ORGANIZATION_BLOCK "MOD_ERR"	// OB 122
TITLE = "Module Access Error"
AUTHOR : Koenig
VERSION : 0.1
VAR_TEMP
  OB122_EV_CLASS : BYTE ;	//16#29, Event class 2, Entering event state, Internal fault event
  OB122_SW_FLT : BYTE ;	//16#XX Software error code
  OB122_PRIORITY : BYTE ;	//Priority of OB Execution
  OB122_OB_NUMBR : BYTE ;	//122 (Organization block 122, OB122)
  OB122_BLK_TYPE : BYTE ;	//16#88/8C/8E Type of block fault occured in
  OB122_MEM_AREA : BYTE ;	//Memory area where access error occured
  OB122_MEM_ADDR : WORD ;	//Memory address where access error occured
  OB122_BLK_NUM : WORD ;	//Block number in which error occured
  OB122_PRG_ADDR : WORD ;	//Program address where error occured
  OB122_DATE_TIME : DATE_AND_TIME ;	//Date and time OB1 started
END_VAR
BEGIN
NETWORK
TITLE =
END_ORGANIZATION_BLOCK

SYMBOL_TABLE
"IDB_Safe_Main"	DB 1	FB 1
"DB_TRO"	DB 2	DB 2
"DB_LIF"	DB 3	DB 3
"DB_TEL"	DB 4	DB 4
"DB_BRI"	DB 5	DB 5
"DB_ComGateway"	DB 10	DB 10
"IDB_FB2_TRO"	DB 12	FB 2
"IDB_FB2_LIF"	DB 13	FB 2
"IDB_FB21_TEL"	DB 14	FB 21
"DB_OrderBuffer"	DB 15	DB 15
"DB_IntentData"	DB 17	DB 17
"DB_TargetData"	DB 19	DB 19
"IDB_FB22"	DB 22	FB 22
"IDB_FB29"	DB 29	FB 29
"IDB_MasterInterface"	DB 33	FB 13
"DB_ANALOG"	DB 50	DB 50
"INOUT"	DB 80	DB 80
"DB_ActualHookdata"	DB 92	DB 92	// Hookdata of actual trollayposition
"Moves"	DB 101	DB 101
"InstanzDB PNIODiag"	DB 126	FB 126
"InstanzDB STATDiag"	DB 127	DB 127
"DB_Crane"	DB 130	DB 130
"DB_Steps"	DB 132	DB 132
"DB_CylinderTypes"	DB 133	DB 133
"DB_Area"	DB 150	DB 150
"IDB_FB190"	DB 190	FB 190
"IDB_FB190_2"	DB 191	FB 190
"IDB1_FB192"	DB 192	FB 192
"IDB1_FB192_2"	DB 193	FB 192
"TRO_Positions"	DB 200	DB 200
"BR01_TR01"	DB 201	DB 201
"BR01_TR02"	DB 202	DB 202
"BR01_TR03"	DB 203	DB 203
"BR01_TR04"	DB 204	DB 204
"BR01_TR05"	DB 205	DB 205
"BR01_TR06"	DB 206	DB 206
"BR01_TR07"	DB 207	DB 207
"BR01_TR08"	DB 208	DB 208
"BR01_TR09"	DB 209	DB 209
"BR01_TR10"	DB 210	DB 210
"BR01_TR11"	DB 211	DB 211
"BR02_TR01"	DB 212	DB 212
"BR02_TR02"	DB 213	DB 213
"BR02_TR03"	DB 214	DB 214
"BR02_TR04"	DB 215	DB 215
"BR02_TR05"	DB 216	DB 216
"BR02_TR06"	DB 217	DB 217
"BR02_TR07"	DB 218	DB 218
"BR02_TR08"	DB 219	DB 219
"BR02_TR09"	DB 220	DB 220
"BR02_TR10"	DB 221	DB 221
"BR02_TR11"	DB 222	DB 222
"BR03_TR01"	DB 223	DB 223
"BR03_TR02"	DB 224	DB 224
"BR03_TR03"	DB 225	DB 225
"BR03_TR04"	DB 226	DB 226
"BR03_TR05"	DB 227	DB 227
"BR03_TR06"	DB 228	DB 228
"BR03_TR07"	DB 229	DB 229
"BR03_TR08"	DB 230	DB 230
"BR03_TR09"	DB 231	DB 231
"BR03_TR10"	DB 232	DB 232
"BR03_TR11"	DB 233	DB 233
"BR04_TR01"	DB 234	DB 234
"BR04_TR02"	DB 235	DB 235
"BR04_TR03"	DB 236	DB 236
"BR04_TR04"	DB 237	DB 237
"BR04_TR05"	DB 238	DB 238
"BR04_TR06"	DB 239	DB 239
"BR04_TR07"	DB 240	DB 240
"BR04_TR08"	DB 241	DB 241
"BR04_TR09"	DB 242	DB 242
"BR04_TR10"	DB 243	DB 243
"BR04_TR11"	DB 244	DB 244
"BR05_TR01"	DB 245	DB 245
"BR05_TR02"	DB 246	DB 246
"BR05_TR03"	DB 247	DB 247
"BR05_TR04"	DB 248	DB 248
"BR05_TR05"	DB 249	DB 249
"BR05_TR06"	DB 250	DB 250
"BR05_TR07"	DB 251	DB 251
"BR05_TR08"	DB 252	DB 252
"BR05_TR09"	DB 253	DB 253
"BR05_TR10"	DB 254	DB 254
"BR05_TR11"	DB 255	DB 255
"BR06_TR01"	DB 256	DB 256
"BR06_TR02"	DB 257	DB 257
"BR06_TR03"	DB 258	DB 258
"BR06_TR04"	DB 259	DB 259
"BR06_TR05"	DB 260	DB 260
"BR06_TR06"	DB 261	DB 261
"BR06_TR07"	DB 262	DB 262
"BR06_TR08"	DB 263	DB 263
"BR06_TR09"	DB 264	DB 264
"BR06_TR10"	DB 265	DB 265
"BR06_TR11"	DB 266	DB 266
"BR07_TR01"	DB 267	DB 267
"BR07_TR02"	DB 268	DB 268
"BR07_TR03"	DB 269	DB 269
"BR07_TR04"	DB 270	DB 270
"BR07_TR05"	DB 271	DB 271
"BR07_TR06"	DB 272	DB 272
"BR07_TR07"	DB 273	DB 273
"BR07_TR08"	DB 274	DB 274
"BR07_TR09"	DB 275	DB 275
"BR07_TR10"	DB 276	DB 276
"BR07_TR11"	DB 277	DB 277
"BR08_TR01"	DB 278	DB 278
"BR08_TR02"	DB 279	DB 279
"BR08_TR03"	DB 280	DB 280
"BR08_TR04"	DB 281	DB 281
"BR08_TR05"	DB 282	DB 282
"BR08_TR06"	DB 283	DB 283
"BR08_TR07"	DB 284	DB 284
"BR08_TR08"	DB 285	DB 285
"BR08_TR09"	DB 286	DB 286
"BR08_TR10"	DB 287	DB 287
"BR08_TR11"	DB 288	DB 288
"BR09_TR01"	DB 289	DB 289
"BR09_TR02"	DB 290	DB 290
"BR09_TR03"	DB 291	DB 291
"BR09_TR04"	DB 292	DB 292
"BR09_TR05"	DB 293	DB 293
"BR09_TR06"	DB 294	DB 294
"BR09_TR07"	DB 295	DB 295
"BR09_TR08"	DB 296	DB 296
"BR09_TR09"	DB 297	DB 297
"BR09_TR10"	DB 298	DB 298
"BR09_TR11"	DB 299	DB 299
"BR10_TR01"	DB 300	DB 300
"BR10_TR02"	DB 301	DB 301
"BR10_TR03"	DB 302	DB 302
"BR10_TR04"	DB 303	DB 303
"BR10_TR05"	DB 304	DB 304
"BR10_TR06"	DB 305	DB 305
"BR10_TR07"	DB 306	DB 306
"BR10_TR08"	DB 307	DB 307
"BR10_TR09"	DB 308	DB 308
"BR10_TR10"	DB 309	DB 309
"BR10_TR11"	DB 310	DB 310
"BR11_TR01"	DB 311	DB 311
"BR11_TR02"	DB 312	DB 312
"LIF_Pos"	DB 350	DB 350
"IDB_Modbus1"	DB 362	FB 102
"ProfiNet"	DB 400	DB 400
"Error_Safety"	DB 410	DB 410
"IDB_ESTOP_1"	DB 450	FB 215
"IDB_ESTOP_2"	DB 451	FB 185
"F_GLOBDB"	DB 545	DB 545	// F_: F_Global_Data Block
"F00035_4FDI_4FDO_iPar__"	DB 555	FB 272
"F00040_4FDI_4FDO_iPar__"	DB 556	FB 272
"F00045_4FDI_iPar___UINT8"	DB 557	FB 272
"F00055_75x_667_4FDI_4FDO"	DB 558	FB 272
"F_IO"	DB 690	DB 690
"F_Position"	DB 695	DB 695
"F_GBL_RECV"	DB 750	DB 750
"IDB_F_RCV"	DB 751	FB 226
"F_GBL_SEND"	DB 752	DB 752
"IDB_F_SND"	DB 753	FB 225
"IDB_Axis_Position"	DB 800	FB 5
"IDB_WagoiPar_Rack"	DB 901	FB 37
"IDB_WagoiPar_BRI"	DB 920	FB 37
"IDB_WagoiPar_TRO"	DB 921	FB 37
"IDB_WagoiPar_LIF"	DB 922	FB 37
"DB_iPar_Diag"	DB 930	FB 101
"DIAG_PROFI_V2_iPar"	DB 931	DB 931	// diagnosis data of PROFIsafe modules V2 iPar with FB101
"DB_Vorlage"	DB 999	DB 999
"DB_LS1"	DB 1300	DB 1300
"IDB_LS1_Circum"	DB 1329	FB 29
"DB_LS"	DB 1350	DB 1350
"iPar_Data_Rack"	DB 1901	DB 1901
"iPar_Data_Bridge"	DB 1920	DB 1920
"iPar_Data_Trolley"	DB 1921	DB 1921
"iPar_Data_Lift"	DB 1922	DB 1922
"Safe_Main"	FB 1	FB 1
"MovidriveB_Control"	FB 2	FB 2
"Axis_Position"	FB 5	FB 5
"MasterInterface"	FB 13	FB 13
"CheckEncoder"	FB 21	FB 21
"GetCircumference"	FB 22	FB 22
"WAGO_Analog_Input_4_20"	FB 29	FB 29	// WAGO A/D-Wandler 4-20mA
"WAGO_iPar_UDL_4_Mod"	FB 37	FB 37	// WAGO up- / download iParameter PROFIsafe Modules
"TSEND"	FB 63	FB 63	// Send Data
"TRCV"	FB 64	FB 64	// Receive Data
"TCON"	FB 65	FB 65	// Connect
"TDISCON"	FB 66	FB 66	// Disconnect
"Safety_Position"	FB 70	FB 70	// Sichere Positionsüberwachung
"Safety_Direction"	FB 72	FB 72	// Sichere Richtungserfassung
"Safety_Speed"	FB 73	FB 73	// Sichere Geschwindigkeit
"Safety_SpeedCheck"	FB 74	FB 74
"Wago_Trolley"	FB 81	FB 81
"F_Input_MAP"	FB 91	FB 91
"ESTOP"	FB 92	FB 92
"GetArea"	FB 95	FB 95
"DiagPROFIsafe_V2_iPar"	FB 101	FB 101	// read diagnosis data of PROFIsafe modules V2 iPar
"MODBUSPN"	FB 102	FB 102	// MODBUS PN CPU
"TCP_COMM"	FB 103	FB 103	// TCP Kommunikation
"MOD_CLI"	FB 104	FB 104
"MOD_SERV"	FB 105	FB 105
"PNIODiag"	FB 126	FB 126	// Profibus/DP und Profinet/IO-Diagnose
"STATDiag"	FB 127	FB 127	// Zweitbaustein (PNIODiag)
"F_TON"	FB 185	FB 185	// F_: Timer Switch On Delay
"F_TOF"	FB 186	FB 186	// F_: Timer Switch Off Delay
"CopyHookDBs"	FB 190	FB 190
"READ_DBL"	FB 192	FB 192	// read db from memorycard
"WRITE_DBL"	FB 193	FB 193	// write db to memorycard
"F_ESTOP1"	FB 215	FB 215	// F_: Emergency Stop / Stop Category 1
"F_ACK_GL"	FB 219	FB 219	// F_: Global Acknowledgement of all F-I/O of a RTG
"F_SENDS7"	FB 225	FB 225	// F_: Send S7 Connection
"F_RCVS7"	FB 226	FB 226	// F_: Receive S7 Connection
"F_IO_CGP"	FB 272	FB 272	// F_: Driver Block In-Output with Channel Granular Passivation
"F_CTRL_1"	FB 273	FB 273
"F_CTRL_2"	FB 274	FB 274	// F_: Test Block an Programm Run Control
"F_DIAG_N"	FB 275	FB 275
"FITON"	FB 276	FB 276
"FITOF"	FB 277	FB 277
"FIACK_GL"	FB 278	FB 278
"F-CALL"	FC 1	FC 1
"Init"	FC 2	FC 2
"AG_SEND"	FC 5	FC 5	// AG SEND
"AG_RECV"	FC 6	FC 6	// AG RECEIVE
"DT_TOD"	FC 8	FC 8	// DT to TOD
"OpHours"	FC 9	FC 9
"EQ_STRNG"	FC 10	FC 10	// Equal String
"AbsEncoder"	FC 11	FC 11
"Motor_2_frequ"	FC 12	FC 12
"DT to DATE"	FC 15	FC 15	// DT to DATE
"Scan_BRI"	FC 21	FC 21
"Scan_BRI_MAN"	FC 22	FC 22	// Scan Bride Manual Mode
"Scan_BRI_DBs"	FC 23	FC 23
"Scan_LIF"	FC 25	FC 25
"Scan_LIF_Man"	FC 26	FC 26
"Scan_TEL"	FC 27	FC 27
"Scan_TEL_Man"	FC 28	FC 28
"SCALE_WAGO_AI"	FC 29	FC 29	// for WAGO 250-466 4-20mA SE Standard
"Inputs"	FC 30	FC 30
"Outputs"	FC 31	FC 31
"MeasureSystem"	FC 33	FC 33
"SEL"	FC 36	FC 36	// Select
"Errors"	FC 40	FC 40
"Errors Reset"	FC 41	FC 41
"Errors_001-016_GEN1"	FC 42	FC 42
"Errors_017-032_GEN2"	FC 43	FC 43
"Errors_033-048_NET"	FC 44	FC 44
"Errors_113-128"	FC 45	FC 45
"Errors_129-144_08"	FC 46	FC 46
"Errors_145-160"	FC 47	FC 47
"EOff_MachineOff"	FC 48	FC 48
"OP_Mode"	FC 49	FC 49
"Send_Buffer"	FC 52	FC 52
"MSG_161-176"	FC 55	FC 55
"MSG_177_192"	FC 56	FC 56
"CableDrum"	FC 60	FC 60
"TargetPosLift"	FC 70	FC 70
"CheckHookType"	FC 72	FC 72
"CheckWindowDi"	FC 100	FC 100
"Communication"	FC 103	FC 103
"STEPS_Control"	FC 110	FC 110
"STEPS_OrderData"	FC 111	FC 111
"STEPS_BASEPOS"	FC 112	FC 112
"STEPS_EMPTY"	FC 113	FC 113
"STEPS_GET"	FC 114	FC 114
"STEPS_PUT"	FC 115	FC 115
"Axis_TROLLEY"	FC 210	FC 210
"Axis_TROLLEY_Release"	FC 211	FC 211
"Axis_TROLLEY_Control"	FC 212	FC 212
"Axis_TROLLEY_Speed"	FC 213	FC 213
"Axis_TROLLEY_Scan"	FC 214	FC 214
"Axis_TROLLEY_Scan_Man"	FC 215	FC 215
"Axis_TROLLEY_Flt_065-080"	FC 219	FC 219
"Axis_LIFT"	FC 220	FC 220
"Axis_LIFT_Control"	FC 222	FC 222
"Axis_LIFT_Speed"	FC 223	FC 223
"Axis_LIFT_Scan"	FC 224	FC 224
"Axis_LIFT_Flt_081-096"	FC 229	FC 229
"Axis_TELESCOPES"	FC 230	FC 230
"Axis_TEL_Control"	FC 232	FC 232
"Axis_TEL_Speed"	FC 233	FC 233
"Axis_TEL_Scan"	FC 234	FC 234
"Axis_TEL_Chk"	FC 235	FC 235
"Axis_TEL_Status"	FC 236	FC 236
"Axis_TEL_Mode_Status"	FC 237	FC 237
"Axis_TEL_BCD"	FC 238	FC 238
"Axis_TEL_Flt_097-112"	FC 239	FC 239
"Axis_TEL_Encoder"	FC 240	FC 240
"iPar_ServerCall"	FC 900	FC 900
"Scan_LIF_New"	FC 1025	FC 1025
"Scan_LIF_Man_New"	FC 1026	FC 1026
"TROGetPosVal"	FC 1071	FC 1071
"E   35.0"	I 35.0	BOOL	// spare
"E   35.1"	I 35.1	BOOL	// spare
"I_TRO_FB_Lift"	I 35.2	BOOL	// Feedback safestop lift
"I_TRO_FB_Trolley"	I 35.3	BOOL	// Feedback safestop  trolley
"I_TRO_FB_Telescope"	I 40.0	BOOL	// Feedback safestop no FU
"E   40.1"	I 40.1	BOOL	// spare
"I_TRO_FB_Estop_CH1"	I 40.2	BOOL	// Feedback E-Stop  CH1
"I_TRO_FB_Estop_CH2"	I 40.3	BOOL	// Feedback E-Stop  CH2
"I_TRO_EStop"	I 45.0	BOOL	// Emergency stop activ
"I_TRO_Brake_OK"	I 45.1	BOOL	// Temperature brake resistors OK
"E   45.2"	I 45.2	BOOL	// spare
"E   45.3"	I 45.3	BOOL	// spare
"I_TRO_LIF_Overl_L_NC"	I 55.0	BOOL	// Overload-Monitoring left NC
"I_TRO_LIF_Overl_R_NC"	I 55.1	BOOL	// Overload-Monitoring right NC
"I_TRO_LIF_Slap_L_NC"	I 55.2	BOOL	// Slap-Rope-Monitoring left NC
"I_TRO_LIF_Slap_R_NC"	I 55.3	BOOL	// Slap-Rope-Monitoring right NC
"I_TRO_Fuse_115V_OK"	I 75.0	BOOL	// 115V AC OK
"I_TRO_Fuse_24V_OK"	I 75.1	BOOL	// fuse 24V DC OK
"I_TRO_Overtemp_Cabinet"	I 75.2	BOOL	// high temperature cabinet
"I_TRO_Power Brakes_OK"	I 75.3	BOOL	// Power supply brakes OK
"I_TRO_Power_Lift_OK"	I 75.4	BOOL	// Power supply lift OK
"I_TRO_Power_Drum_OK"	I 75.5	BOOL	// Power supply cable drum OK
"I_TRO_Power_Cabinet_Fan"	I 75.6	BOOL	// Power supply cabinet fan OK
"I_TRO_Cabinet_Fan_On"	I 75.7	BOOL	// cabinet fan running
"I_TRO_BTN_Reset"	I 76.0	BOOL	// Reset button (top cabinet)
"I_TRO_BTN_Preset"	I 76.1	BOOL	// Preset button (3s)
"I_TRO_Preset_Bit_0"	I 76.2	BOOL	// Preset selection switch bit 0
"I_TRO_Preset_Bit_1"	I 76.3	BOOL	// Preset selection switch bit 1
"I_TRO_Preset_Bit_2"	I 76.4	BOOL	// Preset selection switch bit 2
"I_TRO_Preset_Bit_3"	I 76.5	BOOL	// Preset selection switch bit 3
"E 76_6"	I 76.6	BOOL	// spare
"E 76_7"	I 76.7	BOOL	// spare
"I_Check_CableDrum_NO"	I 77.0	BOOL	// check cable drum NO
"I_Check_CableDrum_NC"	I 77.1	BOOL	// check cable drum NC
"E  77_2"	I 77.2	BOOL	// spar
"E  77_3"	I 77.3	BOOL	// spar
"I_Buffer_left_Free"	I 77.4	BOOL	// Buffer left occupied //
"I_Buffer_right_Free"	I 77.5	BOOL	// Buffer right occupied //
"I_LIF_Limit_TOP"	I 77.6	BOOL	// Lift limit switch top (minus)
"I_LIF_Limit_BOTTOM"	I 77.7	BOOL	// Lift limit switch bottom (plus)
"I_LIF_Pos_TOP_NO"	I 78.0	BOOL	// Lift limit prox. top NO
"I_LIF_Pos_TOP_NC"	I 78.1	BOOL	// Lift limit prox. top NC
"I_TRO_Limit_plus"	I 78.2	BOOL	// Tolley limit switch plus
"I_TRO_Limit_minus"	I 78.3	BOOL	// Tolley limit switch minus
"I_TRO_FS_plus_NO"	I 78.4	BOOL	// Tolley prox. switch forced slow plus NO
"I_TRO_FS_plus_NC"	I 78.5	BOOL	// Tolley prox. switch forced slow plus NC
"I_TRO_FS_minus_NO"	I 78.6	BOOL	// Tolley prox. switch forced slow minus NO
"I_TRO_FS_minus_NC"	I 78.7	BOOL	// Tolley prox. switch forced slow minus NC
"I_SSI_Barcode_noPos"	I 79.0	BOOL	// Datamatrix SSI error: no position
"I_SSI_Barcode_dirty"	I 79.1	BOOL	// Datamatrix SSI error: dirty
"I_Profinet_Barcode_noPos"	I 79.2	BOOL	// Datamatrix Profinet error: no position
"I_Profinet_Barcode_dirty"	I 79.3	BOOL	// Datamatrix Profinet error: dirty
"I_TRO_Drop_1_P"	I 79.4	BOOL	// Trolley drop off protection plus 1
"I_TRO_Drop_2_P"	I 79.5	BOOL	// Trolley drop off protection plus 2
"I_TRO_Drop_1_M"	I 79.6	BOOL	// Trolley drop off protection minus 1
"I_TRO_Drop_2_M"	I 79.7	BOOL	// Trolley drop off protection minus 2
"I_TRO_Plus"	I 80.0	BOOL	// Trolley drive plus
"I_TRO_Minus"	I 80.1	BOOL	// Trolley drive minus
"I_Lift_up"	I 80.2	BOOL	// Lift drive up
"I_Lift_down"	I 80.3	BOOL	// Lift drive down
"I_TEL_Plus"	I 80.4	BOOL	// Tellescope drive plus
"I_TEL_Minus"	I 80.5	BOOL	// Telescope drive minus
"E 80_6"	I 80.6	BOOL	// spare
"E 80_7"	I 80.7	BOOL	// spare
"E 85_0"	I 85.0	BOOL	// spare
"E 85_1"	I 85.1	BOOL	// spare
"E 85_2"	I 85.2	BOOL	// spare
"E 85_3"	I 85.3	BOOL	// spare
"I_TEL_Status1"	I 85.4	BOOL	// Drive telescopes status1
"I_TEL_Status2"	I 85.5	BOOL	// Drive telescopes status2
"E 85_6"	I 85.6	BOOL
"E 85_7"	I 85.7	BOOL
"I_LIF_Overload_L_NO"	I 86.0	BOOL	// Overload-Monitoring left NO
"I_LIF_Overload_R_NO"	I 86.1	BOOL	// Overload-Monitoring right NO
"I_LIF_SlapRope_L_NO"	I 86.2	BOOL	// Slap-Rope-Monitoring left NO
"I_LIF_SlapRope_R_NO"	I 86.3	BOOL	// Slap-Rope-Monitoring right NO
"E      86.4"	I 86.4	BOOL	// spare
"E      86.5"	I 86.5	BOOL	// spare
"I_LIF_Front_LastHookOcc"	I 86.6	BOOL	// hook front left occupied long
"I_LIF_Front_FirstHookOcc"	I 86.7	BOOL	// hook rear left occupied short
"I_LIF_Rear_LastHookOcc"	I 87.0	BOOL	// hook front right occupied long
"I_LIF_Rear_FirstHookOcc"	I 87.1	BOOL	// hook rear right occupied short
"E      87.2"	I 87.2	BOOL	// spare
"E      87.3"	I 87.3	BOOL	// spare
"I_TEL_inMidle_L"	I 87.4	BOOL	// telescope left in middle position
"I_TEL_inMidle_R"	I 87.5	BOOL	// telescope right in middle position
"E      87.6"	I 87.6	BOOL
"I_TEL_Left_Occ_NO"	I 87.7	BOOL	// telescope left occupied NO
"E      88.0"	I 88.0	BOOL
"I_TEL_Right_Occ_NO"	I 88.1	BOOL	// telescope right occupied NO
"I_TEL_Limit_front_NO"	I 88.2	BOOL	// telescopes limit switch front NO
"I_TEL_Limit_front_NC"	I 88.3	BOOL	// telescopes limit switch front NC
"I_TEL_Limit_back_NO"	I 88.4	BOOL	// telescopes limit switch back NO
"I_TEL_Limit_back_NC"	I 88.5	BOOL	// telescopes limit switch back NC
"E      88.6"	I 88.6	BOOL	// spare
"E      88.7"	I 88.7	BOOL	// spare
"E      89.0"	I 89.0	BOOL
"E      89.1"	I 89.1	BOOL
"E      89.2"	I 89.2	BOOL
"E      89.3"	I 89.3	BOOL
"E      89.4"	I 89.4	BOOL
"E      89.5"	I 89.5	BOOL
"E      89.6"	I 89.6	BOOL
"E      89.7"	I 89.7	BOOL
"OFF"	M 0.0	BOOL	// immer aus
"ON"	M 0.1	BOOL	// immer ein
"FIRST_RUN"	M 0.7	BOOL
"ModeService"	M 1.0	BOOL
"ModeManual"	M 1.1	BOOL
"ModeAuto"	M 1.2	BOOL
"ModeBypass"	M 1.3	BOOL
"ModeServiceOrManual"	M 1.4	BOOL
"SEW_EmergencyMode"	M 1.5	BOOL
"ModeAutoOrManual"	M 1.6	BOOL
"LifeBitMasterOK"	M 1.7	BOOL
"Eoff"	M 2.0	BOOL
"DivEoff"	M 2.1	BOOL
"Error"	M 2.2	BOOL
"EmOffRelais_delayed"	M 3.0	BOOL
"TRO_pFL_StopOnCarrier"	M 8.0	BOOL
"TRO_StopOnCarrier"	M 8.1	BOOL
"LIF_pFl_manPrevPos"	M 9.0	BOOL
"LIF_pFl_manNextPos"	M 9.1	BOOL
"Tel_pFl_manMinusPos"	M 9.2	BOOL
"Tel_pFl_manPlusPos"	M 9.3	BOOL
"TEL_nFl_CenterPos"	M 9.4	BOOL
"TEL_StopInCenter"	M 9.5	BOOL
"TEL_pFl_StopInCenter"	M 9.6	BOOL
"Clock0_1"	M 10.0	BOOL	// CPU-Takt 0,1s
"Clock0_2"	M 10.1	BOOL	// CPU-Takt 0,2s
"Clock0_4"	M 10.2	BOOL	// CPU-Takt 0,4s
"Clock0_5"	M 10.3	BOOL	// CPU-Takt 0,5s
"Clock0_8"	M 10.4	BOOL	// CPU-Takt 0,8s
"Clock1_0"	M 10.5	BOOL	// CPU-Takt 1,0s
"Clock1_6"	M 10.6	BOOL	// CPU-Takt 1,6s
"Clock2_0"	M 10.7	BOOL	// CPU-Takt 2,0s
"Tick0_1"	M 11.0	BOOL	// Impuls 0,1s
"Tick0_2"	M 11.1	BOOL	// Impuls 0,2s
"Tick0_4"	M 11.2	BOOL	// Impuls 0,4s
"Tick0_5"	M 11.3	BOOL	// Impuls 0,6s
"Tick0_8"	M 11.4	BOOL	// Impuls 0,8s
"Tick1_0"	M 11.5	BOOL	// Impuls 1,0s
"Tick1_6"	M 11.6	BOOL	// Impuls 1,6s
"Tick2_0"	M 11.7	BOOL	// Impuls 2,0s
"SysPulse_0_1"	M 12.0	BOOL
"SysPulse_0_2"	M 12.1	BOOL
"SysPulse_0_4"	M 12.2	BOOL
"SysPulse_0_5"	M 12.3	BOOL
"SysPulse_0_8"	M 12.4	BOOL
"SysPulse_1_0"	M 12.5	BOOL
"SysPulse_1_6"	M 12.6	BOOL
"SysPulse_2_0"	M 12.7	BOOL
"StartModeAuto"	M 13.0	BOOL
"TEL_pFl_Start"	M 19.0	BOOL
"NullBit"	M 20.0	BOOL
"CB_Lamp_Preset"	M 21.0	BOOL
"TEL_Save_Long_POS_front"	M 25.0	BOOL
"TEL_Save_Long_POS_rear"	M 25.1	BOOL
"TrolleyWasOnCarrier"	M 40.0	BOOL
"SendTrolleyWasOnCarrier"	M 40.1	BOOL
"Next_Step"	M 44.0	BOOL
"SingleStep_ON"	M 44.1	BOOL
"One_Single_Step"	M 44.2	BOOL
"TEL_RackPos"	M 55.0	BOOL
"TEL_LS1_Pos"	M 55.1	BOOL
"TEL_LS2_Pos"	M 55.2	BOOL
"TEL_LS3_Pos"	M 55.3	BOOL
"Safety_Tele_Center"	M 152.0	BOOL
"Safety_Tele_Rear"	M 152.1	BOOL
"Safety_Tele_Front"	M 152.2	BOOL
"Safety_Trolley_in_Pos"	M 153.0	BOOL
"Safety_Lift_Top"	M 154.0	BOOL
"Safety_Lift_Over"	M 154.1	BOOL
"Safety_Lift_Under"	M 154.2	BOOL
"Mode_Bypass"	M 200.2	BOOL
"RED_IBN_Test"	M 420.0	BOOL
"TRUE"	M 500.0	BOOL
"FALSE"	M 500.1	BOOL
"IBN_1"	M 501.0	BOOL
"IBN_0"	M 501.1	BOOL
"IBN_Test"	M 501.2	BOOL
"TRO_iPar_Check"	M 921.0	BOOL
"TRO_iPar_UpLoad"	M 921.1	BOOL
"TRO_iPar_DownL"	M 921.2	BOOL
"TRO_iPar_ReqDiag"	M 921.5	BOOL
"LIF_iPar_Check"	M 922.0	BOOL
"LIF_iPar_UpLoad"	M 922.1	BOOL
"LIF_iPar_DownL"	M 922.2	BOOL
"LIF_iPar_ReqDiag"	M 922.5	BOOL
"TRO_pFl_iPar"	M 925.1	BOOL
"LIF_pFl_iPar_1"	M 925.2	BOOL
"LIF_pFl_iPar_2"	M 925.3	BOOL
"PowerFan_pl"	M 1001.0	BOOL
"PowerFan_n"	M 1001.1	BOOL
"P_FL_TeleCheck1"	M 1401.2	BOOL
"N_FL_TeleCheck1"	M 1401.3	BOOL
"P_FL_TeleCheck2"	M 1401.6	BOOL
"N_FL_TeleCheck2"	M 1401.7	BOOL
"TeleCheckErr1"	M 1402.0	BOOL
"TeleCheckErr2"	M 1402.1	BOOL
"TeleCheckErr3"	M 1402.3	BOOL
"TeleCheckErr4"	M 1402.4	BOOL
"Reset_Err"	M 1410.0	BOOL
"Impuls_1"	M 1500.0	BOOL
"Impuls_2"	M 1500.1	BOOL
"Impuls_3"	M 1500.2	BOOL
"Impuls_4"	M 1500.3	BOOL
"Impuls_5"	M 1500.4	BOOL
"Impuls_6"	M 1500.5	BOOL
"Impuls_7"	M 1500.6	BOOL
"Impuls_8"	M 1500.7	BOOL
"TEL_SaveTarget"	MW 14	INT
"NullWord"	MW 20	WORD
"PC_MSG_Counter"	MW 120	INT
"CYCL_EXC"	OB 1	OB 1
"CYC_INT5"	OB 35	OB 35	// Cyclic Interrupt 5
"CYCL_FLT"	OB 80	OB 80	// Cycle Time Fault
"I/O_FLT1"	OB 82	OB 82	// I/O Point Fault 1
"I/O_FLT2"	OB 83	OB 83	// I/O Point Fault 2
"OBNL_FLT"	OB 85	OB 85	// OB Not Loaded Fault
"RACK_FLT"	OB 86	OB 86	// Loss of Rack Fault
"COMM_FLT"	OB 87	OB 87	// Communication Fault
"STARTUP"	OB 100	OB 100
"PROG_ERR"	OB 121	OB 121	// Programming Error
"MOD_ERR"	OB 122	OB 122	// Module Access Error
"O_Bypass_RC"	Q 35.0	BOOL	// bypass remote control
"A    35.1"	Q 35.1	BOOL	// spare
"O_SafeStop_Lift"	Q 35.2	BOOL	// safe stop lift
"O_SafeStop_Trolley"	Q 35.3	BOOL	// safe stop trolley
"O_SafeStop_Telecope"	Q 40.0	BOOL	// safe stop telescope
"A    40.1"	Q 40.1	BOOL	// spare
"O_TRO_Stop_CH1"	Q 40.2	BOOL	// E-Stop trolley CH1
"O_TRO_Stop_CH2"	Q 40.3	BOOL	// E-Stop trolley CH2
"O_SafeRelease_Telescope"	Q 55.0	BOOL
"A 75_0"	Q 75.0	BOOL	// spare
"O_TRO_Reset_24V"	Q 75.1	BOOL	// reset 24V fuses
"A 75_2"	Q 75.2	BOOL	// spare
"O_TRO_LP_Reset"	Q 75.3	BOOL	// lamp reset
"A 75_4"	Q 75.4	BOOL	// spare
"O_TRO_CableDrum"	Q 75.5	BOOL	// start cable drum
"O_TRO_EStop_Reset"	Q 75.6	BOOL	// ESTOP reset
"O_TRO_LP_Preset"	Q 75.7	BOOL	// lamp preset
"O_TRO_Horn"	Q 76.0	BOOL	// startup warning
"O_TRO_State_0"	Q 76.1	BOOL	// lamp state 0
"O_TRO_State_1"	Q 76.2	BOOL	// lamp state 1
"O_TRO_state_2"	Q 76.3	BOOL	// lamp state 2
"A      76.4"	Q 76.4	BOOL	// spare
"O_TRO_MoviPLC_Reset"	Q 76.5	BOOL	// reset movi PLC
"O_TRO_EmergencyMode"	Q 76.6	BOOL	// Emergency Mode
"O_LIFT_StartFan"	Q 76.7	BOOL	// start Lift Fan
"O_TRO_EmergencyMode_Fwd"	Q 77.0	BOOL	// Emergency mode forward
"O_TRO_EmergencyMode_Bwd"	Q 77.1	BOOL	// Emergency mode backward
"A      77.2"	Q 77.2	BOOL
"A      77.3"	Q 77.3	BOOL
"A      77.4"	Q 77.4	BOOL
"A      77.5"	Q 77.5	BOOL
"A      77.6"	Q 77.6	BOOL
"A      77.7"	Q 77.7	BOOL
"O_TEL_Mode1"	Q 85.0	BOOL	// telescope mode_1 Service
"O_TEL_Mode2"	Q 85.1	BOOL	// telescope mode_2 Automatic
"O_TEL_Start"	Q 85.2	BOOL	// start telescope
"O_TEL_Reset"	Q 85.3	BOOL	// reset telescope
"O_TEL_BCD_Bit_1"	Q 85.4	BOOL	// telescope BCD Bit_1
"O_TEL_BCD_Bit_2"	Q 85.5	BOOL	// telescope BCD Bit_2
"O_TEL_BCD_Bit_3"	Q 85.6	BOOL	// telescope BCD Bit_3
"O_TEL_BCD_Bit_4"	Q 85.7	BOOL	// telescope BCD Bit_4
"O_TEL_LightFront_Left"	Q 86.0	BOOL	// lightning telescopes front left ON
"O_TEL_LightFront_Right"	Q 86.1	BOOL	// lightning telescopes rear rigth ON
"O_TEL_LightRear_Left"	Q 86.2	BOOL	// lightning telescopes rear left ON
"O_TEL_LightRear_Right"	Q 86.3	BOOL	// lightning telescopes rear rigth ON
"O_TEL_Preset_Encoder"	Q 86.4	BOOL	// Preset Encoder Telescope
"A     86.5"	Q 86.5	BOOL	// spare
"A     86.6"	Q 86.6	BOOL	// spare
"A     86.7"	Q 86.7	BOOL	// spare
"A     87.0"	Q 87.0	BOOL
"A     87.1"	Q 87.1	BOOL
"A     87.2"	Q 87.2	BOOL
"A     87.3"	Q 87.3	BOOL
"A     87.4"	Q 87.4	BOOL
"A     87.5"	Q 87.5	BOOL
"A     87.6"	Q 87.6	BOOL
"A     87.7"	Q 87.7	BOOL
"TON"	SFB 4	SFB 4	// Generate an On Delay
"USEND"	SFB 8	SFB 8	// Uncoordinated Sending of Data
"URCV"	SFB 9	SFB 9	// Uncoordinated Receiving of Data
"RDREC"	SFB 52	SFB 52	// Read a Process Data Record
"WRREC"	SFB 53	SFB 53	// Write a Process Data Record
"RALRM"	SFB 54	SFB 54	// Receive Alarm Data
"DPRD_DAT"	SFC 14	SFC 14	// Read Consistent Data of a Standard DP Slave
"DPWR_DAT"	SFC 15	SFC 15	// Write Consistent Data to a Standard DP Slave
"BLKMOV"	SFC 20	SFC 20	// Copy Variables
"FILL"	SFC 21	SFC 21	// Initialize a Memory Area
"TEST_DB"	SFC 24	SFC 24	// Test Data Block
"DIS_AIRT"	SFC 41	SFC 41	// Delay the Higher Priority Interrupts and Asynchronous Errors
"EN_AIRT"	SFC 42	SFC 42	// Enable Higher Priority Interrupts and Asynchronous Errors
"STP"	SFC 46	SFC 46	// Change the CPU to STOP
"RDSYSST"	SFC 51	SFC 51	// Read a System Status List or Partial List
"WR_REC"	SFC 58	SFC 58	// Write Data Record
"RD_REC"	SFC 59	SFC 59	// Read a Data Record
"RD_DBL"	SFC 83	SFC 83	// Read Data Block from Load Memory
"WRIT_DBL"	SFC 84	SFC 84	// Write Data Block in Load Memory
"tPlcOn"	T 1	TIMER
"tAknowl"	T 2	TIMER
"tTimeout_TRO"	T 26	TIMER
"T_TRO_Preset"	T 30	TIMER
"tTimeout_LIF"	T 36	TIMER
"tTimeout_LIF2"	T 37	TIMER
"T_Startup_Warning"	T 94	TIMER
"T_Delay_Emeg_Mode"	T 110	TIMER
"T_Err_TR_Forced_minus"	T 152	TIMER
"T_Err_TR_Forced_plus"	T 153	TIMER
"T_CheckUS"	T 160	TIMER
"T_CheckUS_OK"	T 161	TIMER
"UDT_Any"	UDT 1	UDT 1
"UDT_SysSave"	UDT 2	UDT 2
"OneMove"	UDT 7	UDT 7
"UDT_SEWState"	UDT 11	UDT 11
"UDT_SEWControl"	UDT 12	UDT 12
"TrDataSheet"	UDT 20	UDT 20	// Zuordnung Turm-DBs
"TRODataSheet"	UDT 21	UDT 21
"HookData"	UDT 100	UDT 100
"HookDataSheetNeu"	UDT 101	UDT 101
"HookDataSheet"	UDT 102	UDT 102
"UDT_CylinderType"	UDT 110	UDT 110
"ROW5"	VAT 1	
"IO-Check"	VAT 2	
"ROW4"	VAT 3	
"ROW3"	VAT 4	
"ROW2"	VAT 5	
"ROW1"	VAT 6	
"ROW6"	VAT 7	
"Order"	VAT 8	
"VAT_Sonar"	VAT 9	
"VAT_Bruno"	VAT 10	
"VAT_NewTarget"	VAT 11	
"VAT_TEL_Encoder"	VAT 12	
"VAT_TR_POS_TEST"	VAT 13	
END_SYMBOL_TABLE

TYPE "UDT_Any"	// UDT 1
VERSION : 0.1
  STRUCT
   CONST : BYTE  := B#16#10;	//SIMATIC Constant
   DATATYPE : BYTE ;	//S7-Datatype
   LENGTH : INT ;	//Length of pointer
   DBNO : INT ;	//Datablock Number
   ADDRESS : DWORD ;	//Start address of pointer
  END_STRUCT ;	
END_TYPE

TYPE "UDT_SysSave"	// UDT 2
VERSION : 0.1
  STRUCT
   AR1 : DWORD ;	//adress register 1
   AR2 : DWORD ;	//adress register 2
   DBNO : WORD ;	//DB register
   DINO : WORD ;	//DI register
  END_STRUCT ;	
END_TYPE

TYPE "OneMove"	// UDT 7
VERSION : 0.1
  STRUCT
   MsgCounter : INT ;
   Action : INT ;
   Value_01 : INT ;
   Value_02 : INT ;
   Value_03 : INT ;
   Value_04 : INT ;
   Value_05 : INT ;
   Value_06 : INT ;
   Value_07 : INT ;
   Value_08 : INT ;
   Value_09 : INT ;
   Value_10 : INT ;
   CRC : INT ;
  END_STRUCT ;	
END_TYPE

TYPE "UDT_SEWState"	// UDT 11
VERSION : 0.1
  STRUCT
   State : STRUCT
    Code00 : BOOL ;
    Code01 : BOOL ;
    Code02 : BOOL ;
    Code03 : BOOL ;
    Code04 : BOOL ;
    Code05 : BOOL ;
    Code06 : BOOL ;
    Code07 : BOOL ;
    NgrZero : BOOL ;
    Ready : BOOL ;
    RefOk : BOOL ;
    InPos : BOOL ;
    BrakeOpen : BOOL ;
    ErrWarn : BOOL ;
    LimitRight : BOOL ;
    LimitLeft : BOOL ;
   END_STRUCT ;
   actPosition : DINT ;
   actSpeed : INT ;
   actCurrent : INT ;
   actWorkLoad : INT ;
  END_STRUCT ;	
END_TYPE

TYPE "UDT_SEWControl"	// UDT 12
VERSION : 0.1
  STRUCT
   Control : STRUCT
    Start : BOOL ;
    InchPlus : BOOL ;
    InchMinus : BOOL ;
    Mode11 : BOOL ;
    Mode12 : BOOL ;
    Crt05 : BOOL ;
    Crt06 : BOOL ;
    BypassLimits : BOOL ;
    Lock : BOOL ;
    ReleaseFastStop : BOOL ;
    ReleaseHalt : BOOL ;
    NotPosCrt : BOOL ;
    RampSet2 : BOOL ;
    ParaSet2 : BOOL ;
    Reset : BOOL ;
    Crt17 : BOOL ;
   END_STRUCT ;
   TarPos : DINT ;
   TarSpeed : INT ;
   TarAcc : INT ;
   TarDeac : INT ;
  END_STRUCT ;	
END_TYPE

TYPE "TrDataSheet"	// UDT 20
VERSION : 0.1
  STRUCT
   TroPosVal : DINT ;	//value of trolleyposition
   HookDbNo : INT ;	//number of DB hookdatasheets
  END_STRUCT ;	
END_TYPE

TYPE "TRODataSheet"	// UDT 21
VERSION : 0.1
  STRUCT
   No : INT ;	//number of trolleyposition
   Val : DINT ;	//value of trolleyposition
   HookDbNo : INT ;	//number of DB hookdatasheets
  END_STRUCT ;	
END_TYPE

TYPE "HookData"	// UDT 100
VERSION : 0.1
  STRUCT
   HookType : INT ;
   TotLengthMin : INT ;
   TotLengthMax : INT ;
   FaceLengthMax : INT ;
   CircumMax : INT ;
   TelPos : DINT ;
   Reserve1 : INT ;
  END_STRUCT ;	
END_TYPE

TYPE "HookDataSheetNeu"	// UDT 101
VERSION : 0.1
  STRUCT
   HookOver : DINT ;
   HookUnderOffset : DINT ;
   Telpos_in : DINT ;
   Telpos_mid : DINT ;
   Telpos_out : DINT ;
   TotLengthMin : INT ;
   TotLengthMax : INT ;
   FaceLengthMax : INT ;
   CircumMax : INT ;
   Hooktype : INT ;
   reserve30 : INT ;
  END_STRUCT ;	
END_TYPE

TYPE "HookDataSheet"	// UDT 102
VERSION : 0.1
  STRUCT
   HookOver : DINT ;
   HookUnderOffset : DINT ;
   TelPos_1 : UDT 100;
   TelPos_2 : UDT 100;
   TelPos_3 : UDT 100;
  END_STRUCT ;	
END_TYPE

TYPE "UDT_CylinderType"	// UDT 110
VERSION : 0.1
  STRUCT
   Number : INT ;
   DiameterName : INT ;
   DiameterMin : INT ;
   DiameterMax : INT ;
   Reserve1 : INT ;
  END_STRUCT ;	
END_TYPE

FUNCTION_BLOCK "Safe_Main"	// FB 1
TITLE = Main safety
AUTHOR : Koenig
VERSION : 0.1
VAR
  ON : BOOL ;
  OFF : BOOL ;
  M_Reset : BOOL ;
  M_Automatic : BOOL ;
  StateOK : BOOL ;
  HardwareOK : BOOL ;
  ESTOP : BOOL ;
  ESTOP_DEL : BOOL ;
  Rel_LS : BOOL ;
  Stop_Doors : BOOL ;
  Stop_Doors_DEL : BOOL ;
  Rel_RBG : BOOL ;
  Rel_Trolley : BOOL ;
  Rel_Lift : BOOL ;
  Rel_Telescope : BOOL ;
  ResetGBL : BOOL ;
  RequestGBL : BOOL ;
  SubsGBL : BOOL ;
  Ack : FB 219;
  IO : FB 91;
  E_Stop : FB 92;
  DEL_Doors : FB 185;
  Wago_Trolley_Lift : FB 81;
  TRO_Valid : BOOL ;
  TRO_SafePos : FB 70;
  TRO_SafeAxis : INT ;
  Get_Area : FB 95;
  Difference_Lo : INT ;
  Difference_Hi : INT ;
  TRO_Speed : FB 74;
  TRO_SafeAxis_Speed : INT ;
  TRO_Direction_Plus : BOOL ;
  TRO_Direction_Minus : BOOL ;
  TRO_Direction : FB 72;
  TRO_Direction_Stop : BOOL ;
  Err_SafeSpeed : BOOL ;
  Err_SafeSpeed_Max : BOOL ;
  T_Reset_GBL : FB 185;
  GetArea : FB 95;
END_VAR
BEGIN
// body was compiled from another editor; compiled code not shown
END_FUNCTION_BLOCK

FUNCTION_BLOCK "MovidriveB_Control"	// FB 2
TITLE = MovidriveB_Control
//main control for the SEW controller
//KNOW_HOW_PROTECT 
//
AUTHOR : Koenig
VERSION : 0.1
VAR_INPUT
  StateWord : INT ;
  FastStop : BOOL ;
  Reset : BOOL ;
  Start : BOOL ;
  InchMinus : BOOL ;
  InchPlus : BOOL ;
  ModeService : BOOL ;
  ModeAuto : BOOL ;
  ModeRef : BOOL ;
  Bypass : BOOL ;
  PlcOn : BOOL ;
  Pulse_1_0 : BOOL ;
  Tick_0_1 : BOOL ;
  ActualPosition : DINT ;
  TargetPosition : DINT ;
  TargetPositionNo : INT ;
  LimitPlus : DINT ;
  LimitMinus : DINT ;
  InPosWin : DINT ;
END_VAR
VAR_OUTPUT
  CrtWord : INT ;
  Moves : BOOL ;
  Ready : BOOL ;
  RefOk : BOOL ;
  InPos : BOOL ;
  BrakeOpen : BOOL ;
  Error : BOOL ;
  ErrCode : INT ;
  ActPosition : DINT ;
  ActPositionNo : INT ;
  ActTarget : DINT ;
END_VAR
VAR
  INT_iCntRelHalt : INT ;
  INT_iCntInPos : INT ;
  INT_ActualPosition : DINT ;
  INT_ActualPositionNo : INT ;
  INT_pFl_ResetPosition : BOOL ;
  INT_TargetOK : BOOL ;
END_VAR
VAR_TEMP
  INT_xStateCode00 : BOOL ;
  INT_xStateCode01 : BOOL ;
  INT_xStateCode02 : BOOL ;
  INT_xStateCode03 : BOOL ;
  INT_xStateCode04 : BOOL ;
  INT_xStateCode05 : BOOL ;
  INT_xStateCode06 : BOOL ;
  INT_xStateCode07 : BOOL ;
  INT_xState : BOOL ;
  INT_xStateReady : BOOL ;
  INT_xStateRefOk : BOOL ;
  INT_xStateInPos : BOOL ;
  INT_xStateNgrNull : BOOL ;
  INT_xStateErrWarn : BOOL ;
  INT_xStateLimitRight : BOOL ;
  INT_xStateLimitLeft : BOOL ;
  INT_xCrtStart : BOOL ;
  INT_xCrtInchPlus : BOOL ;
  INT_xCrtInchMinus : BOOL ;
  INT_xCrtMode11 : BOOL ;
  INT_xCrtMode12 : BOOL ;
  INT_xCrt13 : BOOL ;
  INT_xCrt14 : BOOL ;
  INT_xCrtBypassLimits : BOOL ;
  INT_xCrtLock : BOOL ;
  INT_xCrtRelFaststop : BOOL ;
  INT_xCrtRelHalt : BOOL ;
  INT_xCrtNotPosCrt : BOOL ;
  INT_xCrtRampsSet2 : BOOL ;
  INT_xCrtParaSet2 : BOOL ;
  INT_xCrtReset : BOOL ;
  INT_xCrt06 : BOOL ;
  INT_xModeMan : BOOL ;
  INT_xModeAuto : BOOL ;
  INT_xModeRef : BOOL ;
  INT_ON : BOOL ;
  INT_w00 : WORD ;
  mValue : DINT ;
  pValue : DINT ;
END_VAR
BEGIN
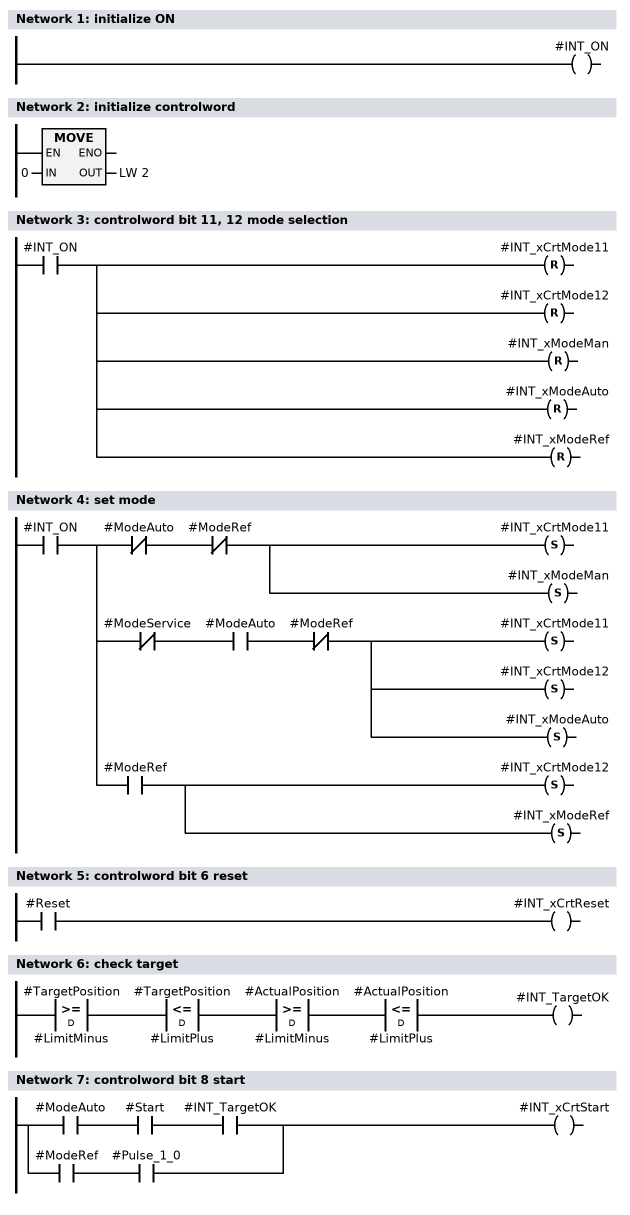
NETWORK
TITLE = initialize ON
//LW0: controler state word
//LW2: controler control word
      SET;
      =     #INT_ON;
NETWORK
TITLE = initialize controlword
      L     0;
      T     LW 2;
      NOP   0;
NETWORK
TITLE = controlword bit 11, 12 mode selection
      A     #INT_ON;
      R     #INT_xCrtMode11;
      R     #INT_xCrtMode12;
      R     #INT_xModeMan;
      R     #INT_xModeAuto;
      R     #INT_xModeRef;
NETWORK
TITLE = set mode
      A     #INT_ON;
      =     L 16.0;
      A     L 16.0;
      AN    #ModeAuto;
      AN    #ModeRef;
      S     #INT_xCrtMode11;
      S     #INT_xModeMan;
      A     L 16.0;
      AN    #ModeService;
      A     #ModeAuto;
      AN    #ModeRef;
      S     #INT_xCrtMode11;
      S     #INT_xCrtMode12;
      S     #INT_xModeAuto;
      A     L 16.0;
      A     #ModeRef;
      S     #INT_xCrtMode12;
      S     #INT_xModeRef;
NETWORK
TITLE = controlword bit 6 reset
      A     #Reset;
      =     #INT_xCrtReset;
NETWORK
TITLE = check target
      A(;
      L     #TargetPosition;
      L     #LimitMinus;
      >=D;
      );
      A(;
      L     #TargetPosition;
      L     #LimitPlus;
      <=D;
      );
      A(;
      L     #ActualPosition;
      L     #LimitMinus;
      >=D;
      );
      A(;
      L     #ActualPosition;
      L     #LimitPlus;
      <=D;
      );
      =     #INT_TargetOK;
NETWORK
TITLE = controlword bit 8 start
      A     #ModeAuto;
      A     #Start;
      A     #INT_TargetOK;
      O;
      A     #ModeRef;
      A     #Pulse_1_0;
      =     #INT_xCrtStart;
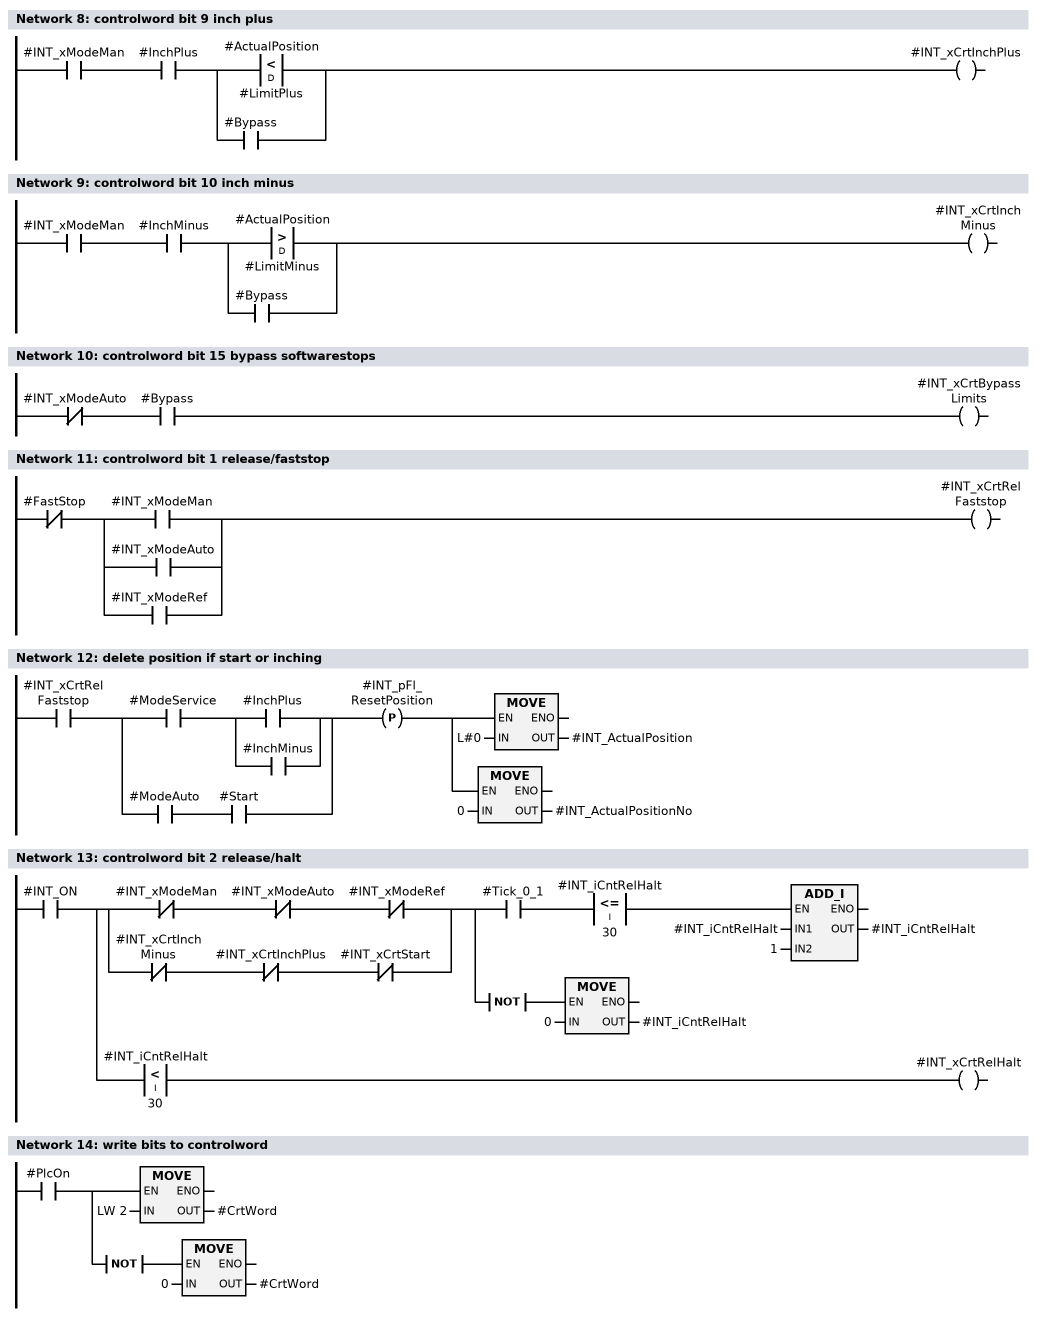
NETWORK
TITLE = controlword bit 9 inch plus
      A     #INT_xModeMan;
      A     #InchPlus;
      A(;
      O(;
      L     #ActualPosition;
      L     #LimitPlus;
      <D;
      );
      O     #Bypass;
      );
      =     #INT_xCrtInchPlus;
NETWORK
TITLE = controlword bit 10 inch minus
      A     #INT_xModeMan;
      A     #InchMinus;
      A(;
      O(;
      L     #ActualPosition;
      L     #LimitMinus;
      >D;
      );
      O     #Bypass;
      );
      =     #INT_xCrtInchMinus;
NETWORK
TITLE = controlword bit 15 bypass softwarestops
      AN    #INT_xModeAuto;
      A     #Bypass;
      =     #INT_xCrtBypassLimits;
NETWORK
TITLE = controlword bit 1 release/faststop
      AN    #FastStop;
      A(;
      O     #INT_xModeMan;
      O     #INT_xModeAuto;
      O     #INT_xModeRef;
      );
      =     #INT_xCrtRelFaststop;
NETWORK
TITLE = delete position if start or inching
      A     #INT_xCrtRelFaststop;
      A(;
      A     #ModeService;
      A(;
      O     #InchPlus;
      O     #InchMinus;
      );
      O;
      A     #ModeAuto;
      A     #Start;
      );
      FP    #INT_pFl_ResetPosition;
      =     L 16.0;
      A     L 16.0;
      JNB   _001;
      L     L#0;
      T     #INT_ActualPosition;
_001: NOP   0;
      A     L 16.0;
      JNB   _002;
      L     0;
      T     #INT_ActualPositionNo;
_002: NOP   0;
NETWORK
TITLE = controlword bit 2 release/halt
      A     #INT_ON;
      =     L 16.0;
      A     L 16.0;
      A(;
      AN    #INT_xModeMan;
      AN    #INT_xModeAuto;
      AN    #INT_xModeRef;
      O;
      AN    #INT_xCrtInchMinus;
      AN    #INT_xCrtInchPlus;
      AN    #INT_xCrtStart;
      );
      =     L 16.1;
      A     L 16.1;
      A     #Tick_0_1;
      A(;
      L     #INT_iCntRelHalt;
      L     30;
      <=I;
      );
      JNB   _003;
      L     #INT_iCntRelHalt;
      L     1;
      +I;
      T     #INT_iCntRelHalt;
_003: NOP   0;
      A     L 16.1;
      NOT;
      JNB   _004;
      L     0;
      T     #INT_iCntRelHalt;
_004: NOP   0;
      A     L 16.0;
      A(;
      L     #INT_iCntRelHalt;
      L     30;
      <I;
      );
      =     #INT_xCrtRelHalt;
NETWORK
TITLE = write bits to controlword
      A     #PlcOn;
      =     L 16.0;
      A     L 16.0;
      JNB   _005;
      L     LW 2;
      T     #CrtWord;
_005: NOP   0;
      A     L 16.0;
      NOT;
      JNB   _006;
      L     0;
      T     #CrtWord;
_006: NOP   0;
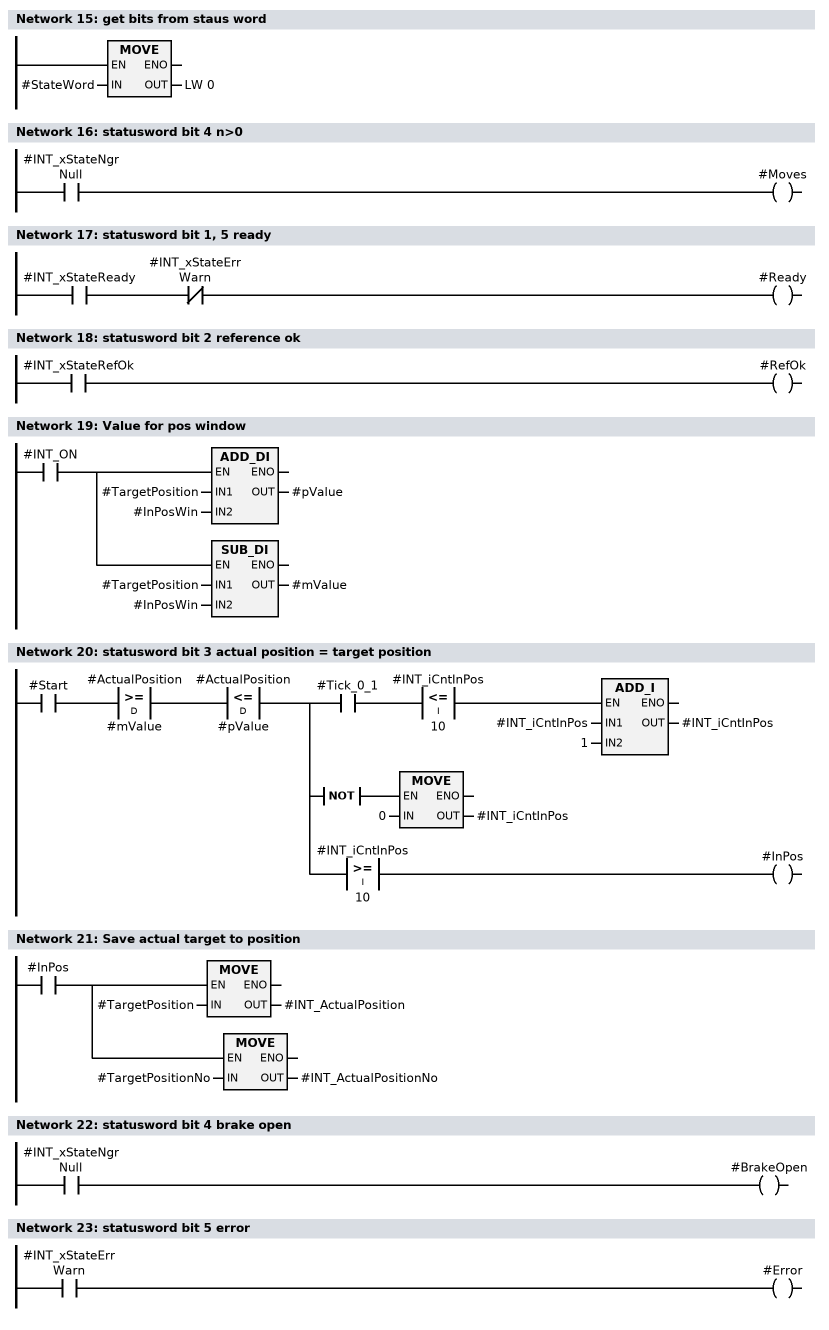
NETWORK
TITLE = get bits from staus word
      L     #StateWord;
      T     LW 0;
      NOP   0;
NETWORK
TITLE = statusword bit 4 n>0
      A     #INT_xStateNgrNull;
      =     #Moves;
NETWORK
TITLE = statusword bit 1, 5 ready
      A     #INT_xStateReady;
      AN    #INT_xStateErrWarn;
      =     #Ready;
NETWORK
TITLE = statusword bit 2 reference ok
      A     #INT_xStateRefOk;
      =     #RefOk;
NETWORK
TITLE = Value for pos window
      A     #INT_ON;
      =     L 16.0;
      A     L 16.0;
      JNB   _007;
      L     #TargetPosition;
      L     #InPosWin;
      +D;
      T     #pValue;
_007: NOP   0;
      A     L 16.0;
      JNB   _008;
      L     #TargetPosition;
      L     #InPosWin;
      -D;
      T     #mValue;
_008: NOP   0;
NETWORK
TITLE = statusword bit 3 actual position = target position
//note: in omron we use the actual position and the target postion equal
//
      A     #Start;
      A(;
      L     #ActualPosition;
      L     #mValue;
      >=D;
      );
      A(;
      L     #ActualPosition;
      L     #pValue;
      <=D;
      );
      =     L 16.0;
      A     L 16.0;
      A     #Tick_0_1;
      A(;
      L     #INT_iCntInPos;
      L     10;
      <=I;
      );
      JNB   _009;
      L     #INT_iCntInPos;
      L     1;
      +I;
      T     #INT_iCntInPos;
_009: NOP   0;
      A     L 16.0;
      NOT;
      JNB   _00a;
      L     0;
      T     #INT_iCntInPos;
_00a: NOP   0;
      A     L 16.0;
      A(;
      L     #INT_iCntInPos;
      L     10;
      >=I;
      );
      =     #InPos;
NETWORK
TITLE = Save actual target to position
      A     #InPos;
      =     L 16.0;
      A     L 16.0;
      JNB   _00b;
      L     #TargetPosition;
      T     #INT_ActualPosition;
_00b: NOP   0;
      A     L 16.0;
      JNB   _00c;
      L     #TargetPositionNo;
      T     #INT_ActualPositionNo;
_00c: NOP   0;
NETWORK
TITLE = statusword bit 4 brake open
      A     #INT_xStateNgrNull;
      =     #BrakeOpen;
NETWORK
TITLE = statusword bit 5 error
      A     #INT_xStateErrWarn;
      =     #Error;
NETWORK
TITLE = status / error code
      A     #INT_ON;
      =     L 16.0;
      A     L 16.0;
      JNB   _00d;
      L     LW 0;
      L     W#16#FF00;
      AW;
      T     LW 0;
_00d: NOP   0;
      A     L 16.0;
      JNB   _00e;
      L     W#16#8;
      L     LW 0;
      SRW;
      T     LW 0;
_00e: NOP   0;
      A     L 16.0;
      JNB   _00f;
      L     LW 0;
      T     #ErrCode;
_00f: NOP   0;
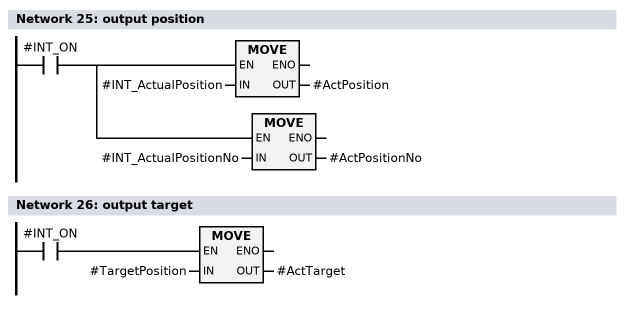
NETWORK
TITLE = output position
      A     #INT_ON;
      =     L 16.0;
      A     L 16.0;
      JNB   _010;
      L     #INT_ActualPosition;
      T     #ActPosition;
_010: NOP   0;
      A     L 16.0;
      JNB   _011;
      L     #INT_ActualPositionNo;
      T     #ActPositionNo;
_011: NOP   0;
NETWORK
TITLE = output target
      A     #INT_ON;
      JNB   _012;
      L     #TargetPosition;
      T     #ActTarget;
_012: NOP   0;
END_FUNCTION_BLOCK

FUNCTION_BLOCK "Axis_Position"	// FB 5
TITLE = Axis_Position
AUTHOR : BRO
VERSION : 0.1
VAR_INPUT
  Inpos : DINT ;
END_VAR
VAR_OUTPUT
  OutPos : DINT ;
END_VAR
BEGIN
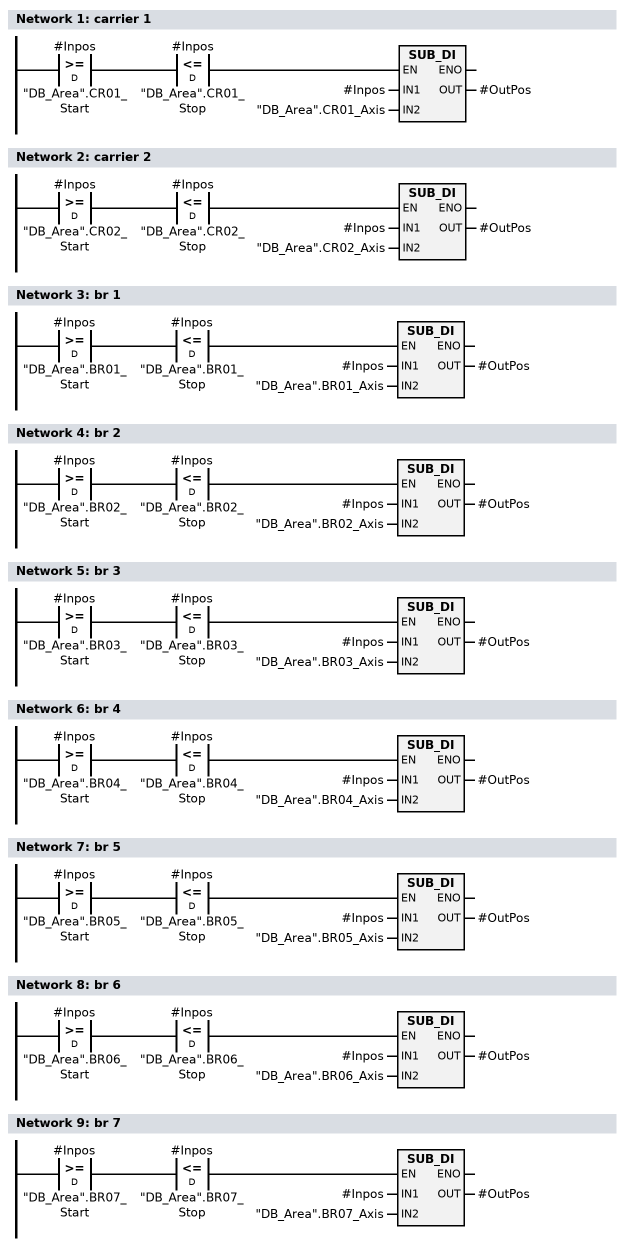
NETWORK
TITLE = carrier 1
      A(;
      L     #Inpos;
      L     "DB_Area".CR01_Start;
      >=D;
      );
      A(;
      L     #Inpos;
      L     "DB_Area".CR01_Stop;
      <=D;
      );
      JNB   _001;
      L     #Inpos;
      L     "DB_Area".CR01_Axis;
      -D;
      T     #OutPos;
_001: NOP   0;
NETWORK
TITLE = carrier 2
      A(;
      L     #Inpos;
      L     "DB_Area".CR02_Start;
      >=D;
      );
      A(;
      L     #Inpos;
      L     "DB_Area".CR02_Stop;
      <=D;
      );
      JNB   _002;
      L     #Inpos;
      L     "DB_Area".CR02_Axis;
      -D;
      T     #OutPos;
_002: NOP   0;
NETWORK
TITLE = br 1
      A(;
      L     #Inpos;
      L     "DB_Area".BR01_Start;
      >=D;
      );
      A(;
      L     #Inpos;
      L     "DB_Area".BR01_Stop;
      <=D;
      );
      JNB   _003;
      L     #Inpos;
      L     "DB_Area".BR01_Axis;
      -D;
      T     #OutPos;
_003: NOP   0;
NETWORK
TITLE = br 2
      A(;
      L     #Inpos;
      L     "DB_Area".BR02_Start;
      >=D;
      );
      A(;
      L     #Inpos;
      L     "DB_Area".BR02_Stop;
      <=D;
      );
      JNB   _004;
      L     #Inpos;
      L     "DB_Area".BR02_Axis;
      -D;
      T     #OutPos;
_004: NOP   0;
NETWORK
TITLE = br 3
      A(;
      L     #Inpos;
      L     "DB_Area".BR03_Start;
      >=D;
      );
      A(;
      L     #Inpos;
      L     "DB_Area".BR03_Stop;
      <=D;
      );
      JNB   _005;
      L     #Inpos;
      L     "DB_Area".BR03_Axis;
      -D;
      T     #OutPos;
_005: NOP   0;
NETWORK
TITLE = br 4
      A(;
      L     #Inpos;
      L     "DB_Area".BR04_Start;
      >=D;
      );
      A(;
      L     #Inpos;
      L     "DB_Area".BR04_Stop;
      <=D;
      );
      JNB   _006;
      L     #Inpos;
      L     "DB_Area".BR04_Axis;
      -D;
      T     #OutPos;
_006: NOP   0;
NETWORK
TITLE = br 5
      A(;
      L     #Inpos;
      L     "DB_Area".BR05_Start;
      >=D;
      );
      A(;
      L     #Inpos;
      L     "DB_Area".BR05_Stop;
      <=D;
      );
      JNB   _007;
      L     #Inpos;
      L     "DB_Area".BR05_Axis;
      -D;
      T     #OutPos;
_007: NOP   0;
NETWORK
TITLE = br 6
      A(;
      L     #Inpos;
      L     "DB_Area".BR06_Start;
      >=D;
      );
      A(;
      L     #Inpos;
      L     "DB_Area".BR06_Stop;
      <=D;
      );
      JNB   _008;
      L     #Inpos;
      L     "DB_Area".BR06_Axis;
      -D;
      T     #OutPos;
_008: NOP   0;
NETWORK
TITLE = br 7
      A(;
      L     #Inpos;
      L     "DB_Area".BR07_Start;
      >=D;
      );
      A(;
      L     #Inpos;
      L     "DB_Area".BR07_Stop;
      <=D;
      );
      JNB   _009;
      L     #Inpos;
      L     "DB_Area".BR07_Axis;
      -D;
      T     #OutPos;
_009: NOP   0;
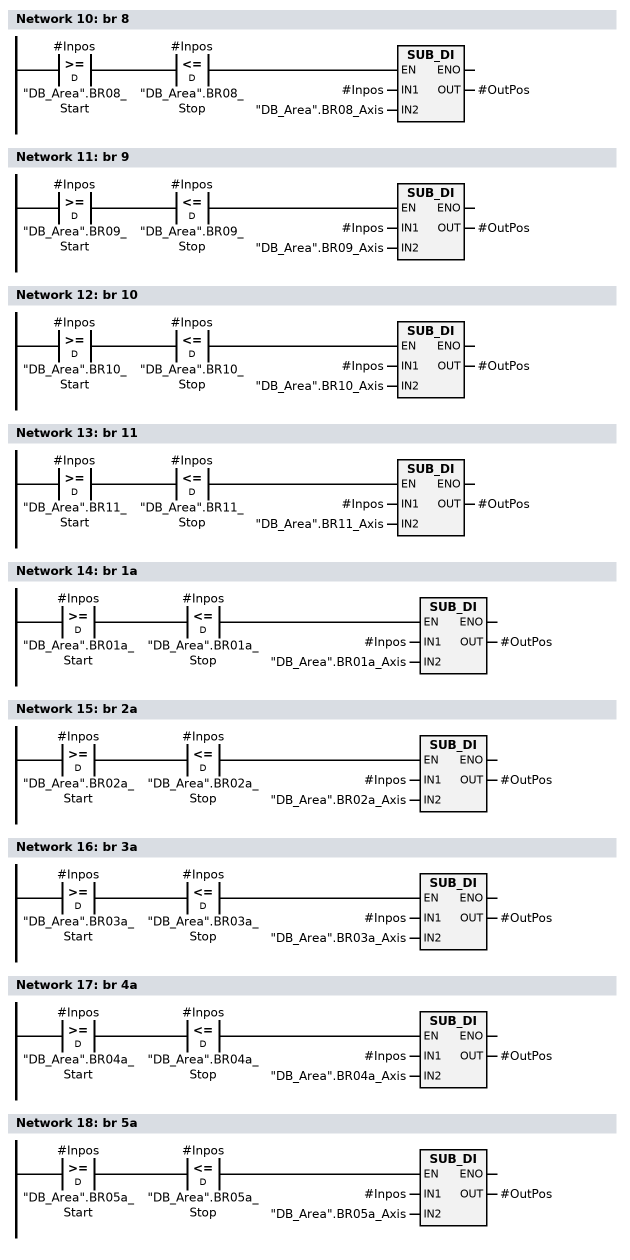
NETWORK
TITLE = br 8
      A(;
      L     #Inpos;
      L     "DB_Area".BR08_Start;
      >=D;
      );
      A(;
      L     #Inpos;
      L     "DB_Area".BR08_Stop;
      <=D;
      );
      JNB   _00a;
      L     #Inpos;
      L     "DB_Area".BR08_Axis;
      -D;
      T     #OutPos;
_00a: NOP   0;
NETWORK
TITLE = br 9
      A(;
      L     #Inpos;
      L     "DB_Area".BR09_Start;
      >=D;
      );
      A(;
      L     #Inpos;
      L     "DB_Area".BR09_Stop;
      <=D;
      );
      JNB   _00b;
      L     #Inpos;
      L     "DB_Area".BR09_Axis;
      -D;
      T     #OutPos;
_00b: NOP   0;
NETWORK
TITLE = br 10
      A(;
      L     #Inpos;
      L     "DB_Area".BR10_Start;
      >=D;
      );
      A(;
      L     #Inpos;
      L     "DB_Area".BR10_Stop;
      <=D;
      );
      JNB   _00c;
      L     #Inpos;
      L     "DB_Area".BR10_Axis;
      -D;
      T     #OutPos;
_00c: NOP   0;
NETWORK
TITLE = br 11
      A(;
      L     #Inpos;
      L     "DB_Area".BR11_Start;
      >=D;
      );
      A(;
      L     #Inpos;
      L     "DB_Area".BR11_Stop;
      <=D;
      );
      JNB   _00d;
      L     #Inpos;
      L     "DB_Area".BR11_Axis;
      -D;
      T     #OutPos;
_00d: NOP   0;
NETWORK
TITLE = br 1a
      A(;
      L     #Inpos;
      L     "DB_Area".BR01a_Start;
      >=D;
      );
      A(;
      L     #Inpos;
      L     "DB_Area".BR01a_Stop;
      <=D;
      );
      JNB   _00e;
      L     #Inpos;
      L     "DB_Area".BR01a_Axis;
      -D;
      T     #OutPos;
_00e: NOP   0;
NETWORK
TITLE = br 2a
      A(;
      L     #Inpos;
      L     "DB_Area".BR02a_Start;
      >=D;
      );
      A(;
      L     #Inpos;
      L     "DB_Area".BR02a_Stop;
      <=D;
      );
      JNB   _00f;
      L     #Inpos;
      L     "DB_Area".BR02a_Axis;
      -D;
      T     #OutPos;
_00f: NOP   0;
NETWORK
TITLE = br 3a
      A(;
      L     #Inpos;
      L     "DB_Area".BR03a_Start;
      >=D;
      );
      A(;
      L     #Inpos;
      L     "DB_Area".BR03a_Stop;
      <=D;
      );
      JNB   _010;
      L     #Inpos;
      L     "DB_Area".BR03a_Axis;
      -D;
      T     #OutPos;
_010: NOP   0;
NETWORK
TITLE = br 4a
      A(;
      L     #Inpos;
      L     "DB_Area".BR04a_Start;
      >=D;
      );
      A(;
      L     #Inpos;
      L     "DB_Area".BR04a_Stop;
      <=D;
      );
      JNB   _011;
      L     #Inpos;
      L     "DB_Area".BR04a_Axis;
      -D;
      T     #OutPos;
_011: NOP   0;
NETWORK
TITLE = br 5a
      A(;
      L     #Inpos;
      L     "DB_Area".BR05a_Start;
      >=D;
      );
      A(;
      L     #Inpos;
      L     "DB_Area".BR05a_Stop;
      <=D;
      );
      JNB   _012;
      L     #Inpos;
      L     "DB_Area".BR05a_Axis;
      -D;
      T     #OutPos;
_012: NOP   0;
END_FUNCTION_BLOCK

FUNCTION_BLOCK "MasterInterface"	// FB 13
//LW0: control word from master
//LW2: status word to master
VERSION : 0.1
VAR_INPUT
  IN_iCrtWord : INT ;
  IN_iCommCounter : INT ;
  IN_iToggleTime_0_1sec : INT ;
  IN_xFree : BOOL ;
  IN_xOccupied : BOOL ;
  IN_xLiftTop : BOOL ;
  IN_xOnline : BOOL ;
  IN_xReadyOnline : BOOL ;
  IN_xError : BOOL ;
  IN_xMovingSource : BOOL ;
  IN_xMovingTarget : BOOL ;
  IN_x09 : BOOL ;
  IN_xOrderRunning : BOOL ;
  IN_xOrderEnd : BOOL ;
  IN_xOrderPaused : BOOL ;
  IN_x13 : BOOL ;
  IN_xNewTarget : BOOL ;
  IN_x15 : BOOL ;
  IN_SysTick : BOOL ;
END_VAR
VAR_OUTPUT
  OUT_iStateWord : INT ;
  OUT_xLifeBitOk : BOOL ;
  OUT_x01 : BOOL ;
  OUT_xStartBasePos : BOOL ;
  OUT_xStartNewTarget : BOOL ;
  OUT_xAknOrderEnd : BOOL ;
  OUT_xReset : BOOL ;
  OUT_x06 : BOOL ;
  OUT_x07 : BOOL ;
  OUT_x08 : BOOL ;
  OUT_x09 : BOOL ;
  OUT_xStartOrder : BOOL ;
  OUT_xClearOrder : BOOL ;
  OUT_xPauseOrder : BOOL ;
  OUT_x13 : BOOL ;
  OUT_xStartStopPos : BOOL ;
  OUT_xReleaseOnline : BOOL ;
END_VAR
VAR
  INT_b_1 : BOOL ;
  INT_b_2 : BOOL ;
  INT_b_3 : BOOL ;
  INT_iCntLbOn : INT ;
  INT_iCntLbOff : INT ;
  INT_iCntLbOk : INT ;
  INT_iCntStartBasePos : INT ;
  INT_iCntStartNewtarget : INT ;
  INT_iCntStartOrder : INT ;
  INT_iCntStartStopPos : INT ;
  INT_iLastCommCounter : INT ;
  INT_T1 : SFB 4;
  INT_T2 : SFB 4;
END_VAR
VAR_TEMP
  INT_xCrt08 : BOOL ;
  INT_xCrt09 : BOOL ;
  INT_xCrtStartOrder : BOOL ;
  INT_xCrtClearOrder : BOOL ;
  INT_xCrtPauseOrder : BOOL ;
  INT_xCrt13 : BOOL ;
  INT_xCrtStartStopPos : BOOL ;
  INT_xReleaseOnline : BOOL ;
  INT_xCrtLife : BOOL ;
  INT_xCrt01 : BOOL ;
  INT_xCrtStartBasePos : BOOL ;
  INT_xCrtStartNewTarg : BOOL ;
  INT_xCrtAcknOrderEnd : BOOL ;
  INT_xCrtReset : BOOL ;
  INT_xCrt06 : BOOL ;
  INT_xCrt07 : BOOL ;
  INT_xStateMovingTarget : BOOL ;
  INT_xState09 : BOOL ;
  INT_xStateOrderRunning : BOOL ;
  INT_xStateOrderEnd : BOOL ;
  INT_xStateOrderPaused : BOOL ;
  INT_xState13 : BOOL ;
  INT_xStateNewTarget : BOOL ;
  INT_xState15 : BOOL ;
  INT_xStateLife : BOOL ;
  INT_xStateFree : BOOL ;
  INT_xStateOccupied : BOOL ;
  INT_xStateLiftTop : BOOL ;
  INT_xStateOnline : BOOL ;
  INT_xStateReadyOnline : BOOL ;
  INT_xStateError : BOOL ;
  INT_xStateMovingSource : BOOL ;
  ON : BOOL ;
END_VAR
BEGIN
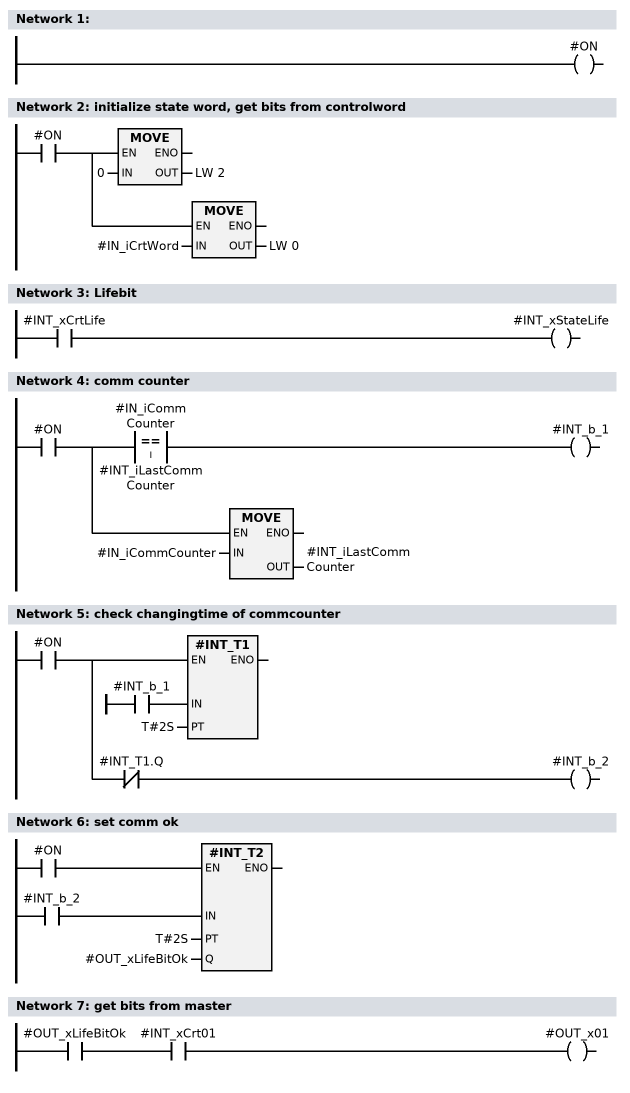
NETWORK
TITLE =
      SET;
      =     #ON;
NETWORK
TITLE = initialize state word, get bits from controlword
      A     #ON;
      =     L 5.0;
      A     L 5.0;
      JNB   _001;
      L     0;
      T     LW 2;
_001: NOP   0;
      A     L 5.0;
      JNB   _002;
      L     #IN_iCrtWord;
      T     LW 0;
_002: NOP   0;
NETWORK
TITLE = Lifebit
      A     #INT_xCrtLife;
      =     #INT_xStateLife;
NETWORK
TITLE = comm counter
      A     #ON;
      =     L 5.0;
      A     L 5.0;
      A(;
      L     #IN_iCommCounter;
      L     #INT_iLastCommCounter;
      ==I;
      );
      =     #INT_b_1;
      A     L 5.0;
      JNB   _003;
      L     #IN_iCommCounter;
      T     #INT_iLastCommCounter;
_003: NOP   0;
NETWORK
TITLE = check changingtime of commcounter
      A     #ON;
      =     L 5.0;
      A     #INT_b_1;
      =     L 5.1;
      BLD   103;
      A     L 5.0;
      JNB   _004;
      CALL  #INT_T1 (
           IN                       := L 5.1,
           PT                       := T#2S);
_004: NOP   0;
      A     L 5.0;
      AN    #INT_T1.Q;
      =     #INT_b_2;
NETWORK
TITLE = set comm ok
      A     #INT_b_2;
      =     L 5.0;
      BLD   103;
      A     #ON;
      JNB   _005;
      CALL  #INT_T2 (
           IN                       := L 5.0,
           PT                       := T#2S,
           Q                        := #OUT_xLifeBitOk);
_005: NOP   0;
NETWORK
TITLE = get bits from master
      A     #OUT_xLifeBitOk;
      A     #INT_xCrt01;
      =     #OUT_x01;
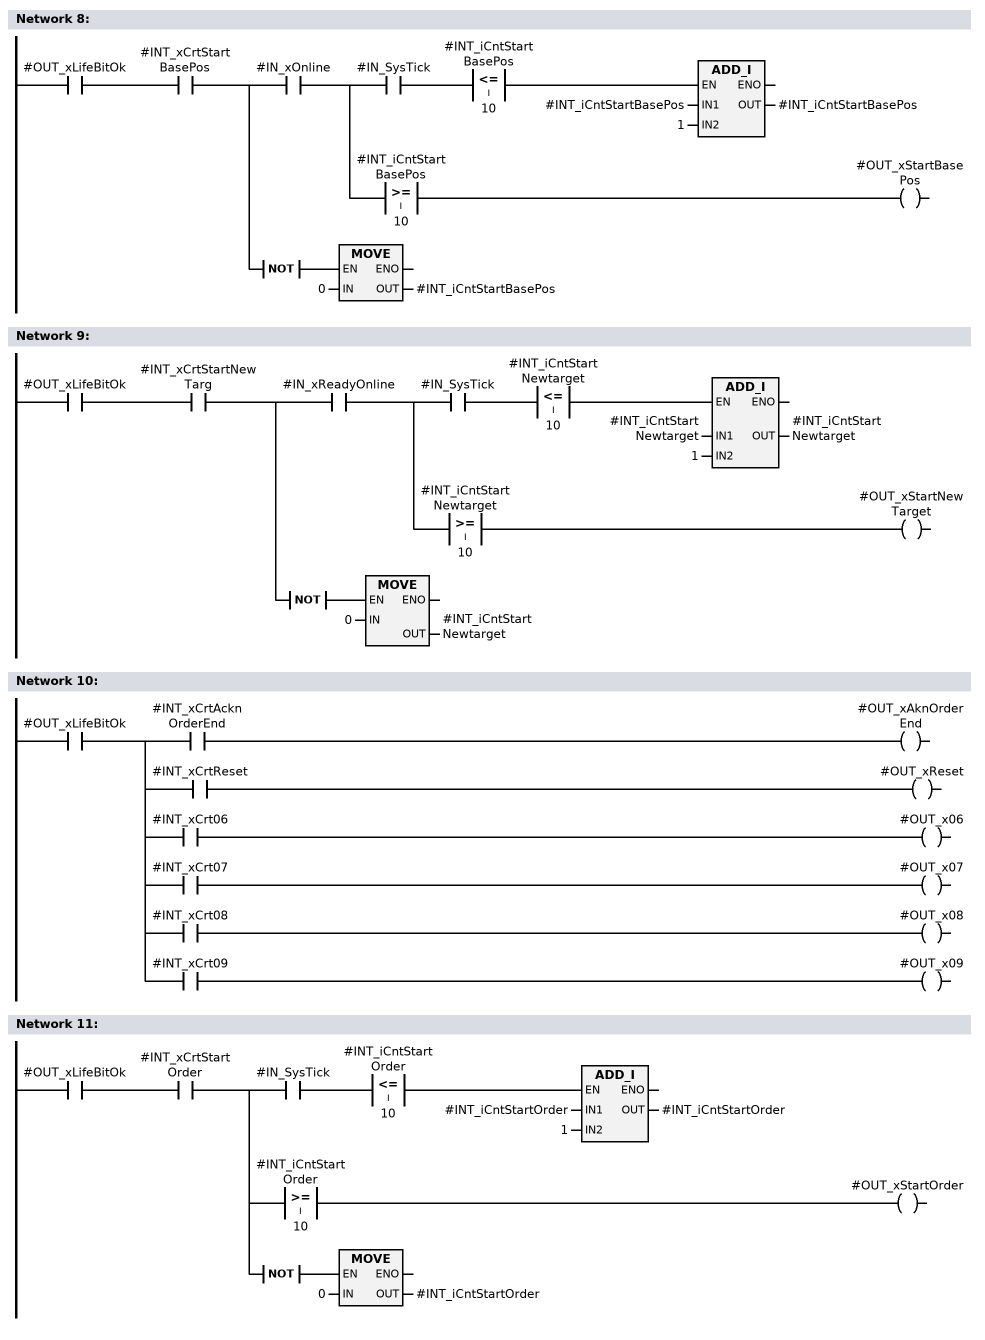
NETWORK
TITLE =
      A     #OUT_xLifeBitOk;
      A     #INT_xCrtStartBasePos;
      =     L 5.0;
      A     L 5.0;
      A     #IN_xOnline;
      =     L 5.1;
      A     L 5.1;
      A     #IN_SysTick;
      A(;
      L     #INT_iCntStartBasePos;
      L     10;
      <=I;
      );
      JNB   _006;
      L     #INT_iCntStartBasePos;
      L     1;
      +I;
      T     #INT_iCntStartBasePos;
_006: NOP   0;
      A     L 5.1;
      A(;
      L     #INT_iCntStartBasePos;
      L     10;
      >=I;
      );
      =     #OUT_xStartBasePos;
      A     L 5.0;
      NOT;
      JNB   _007;
      L     0;
      T     #INT_iCntStartBasePos;
_007: NOP   0;
NETWORK
TITLE =
      A     #OUT_xLifeBitOk;
      A     #INT_xCrtStartNewTarg;
      =     L 5.0;
      A     L 5.0;
      A     #IN_xReadyOnline;
      =     L 5.1;
      A     L 5.1;
      A     #IN_SysTick;
      A(;
      L     #INT_iCntStartNewtarget;
      L     10;
      <=I;
      );
      JNB   _008;
      L     #INT_iCntStartNewtarget;
      L     1;
      +I;
      T     #INT_iCntStartNewtarget;
_008: NOP   0;
      A     L 5.1;
      A(;
      L     #INT_iCntStartNewtarget;
      L     10;
      >=I;
      );
      =     #OUT_xStartNewTarget;
      A     L 5.0;
      NOT;
      JNB   _009;
      L     0;
      T     #INT_iCntStartNewtarget;
_009: NOP   0;
NETWORK
TITLE =
      A     #OUT_xLifeBitOk;
      =     L 5.0;
      A     L 5.0;
      A     #INT_xCrtAcknOrderEnd;
      =     #OUT_xAknOrderEnd;
      A     L 5.0;
      A     #INT_xCrtReset;
      =     #OUT_xReset;
      A     L 5.0;
      A     #INT_xCrt06;
      =     #OUT_x06;
      A     L 5.0;
      A     #INT_xCrt07;
      =     #OUT_x07;
      A     L 5.0;
      A     #INT_xCrt08;
      =     #OUT_x08;
      A     L 5.0;
      A     #INT_xCrt09;
      =     #OUT_x09;
NETWORK
TITLE =
      A     #OUT_xLifeBitOk;
      A     #INT_xCrtStartOrder;
      =     L 5.0;
      A     L 5.0;
      A     #IN_SysTick;
      A(;
      L     #INT_iCntStartOrder;
      L     10;
      <=I;
      );
      JNB   _00a;
      L     #INT_iCntStartOrder;
      L     1;
      +I;
      T     #INT_iCntStartOrder;
_00a: NOP   0;
      A     L 5.0;
      A(;
      L     #INT_iCntStartOrder;
      L     10;
      >=I;
      );
      =     #OUT_xStartOrder;
      A     L 5.0;
      NOT;
      JNB   _00b;
      L     0;
      T     #INT_iCntStartOrder;
_00b: NOP   0;
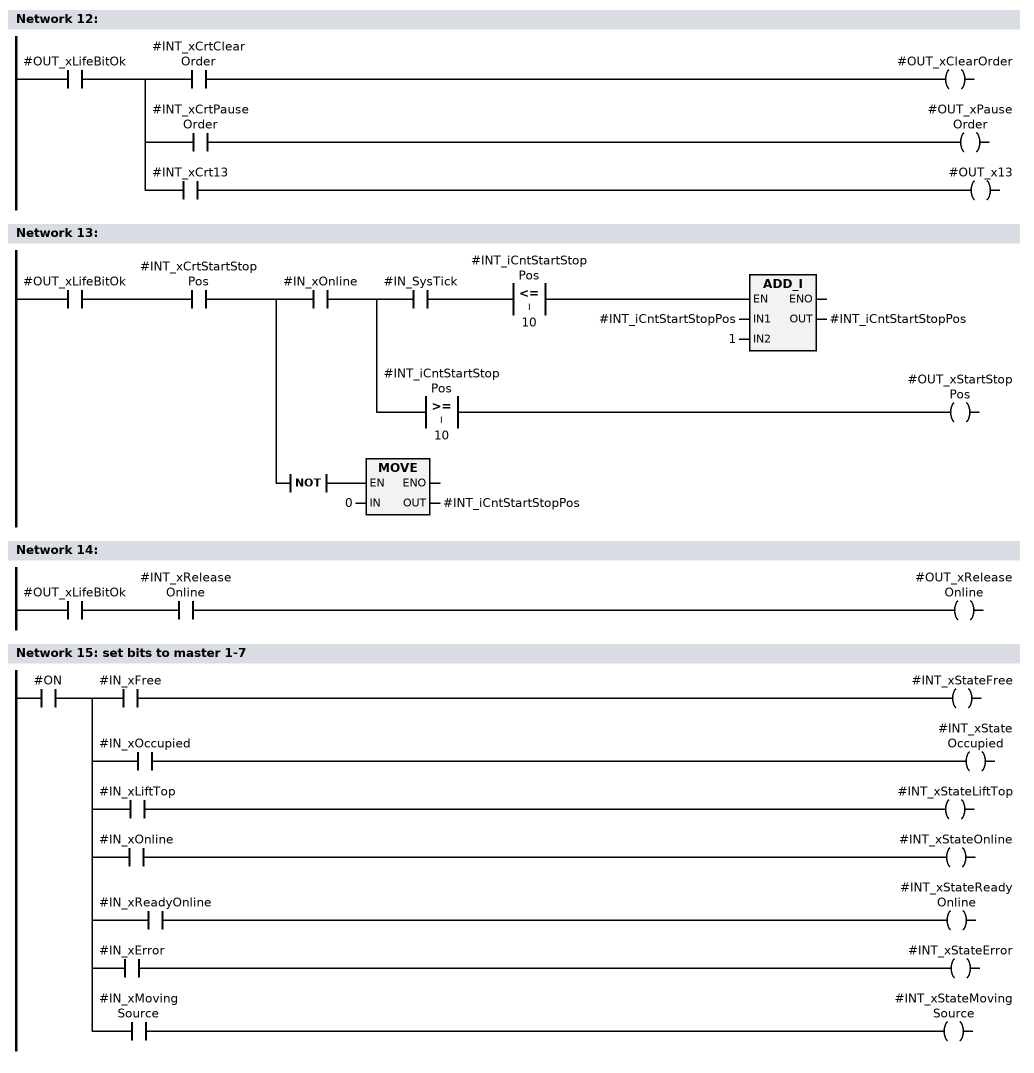
NETWORK
TITLE =
      A     #OUT_xLifeBitOk;
      =     L 5.0;
      A     L 5.0;
      A     #INT_xCrtClearOrder;
      =     #OUT_xClearOrder;
      A     L 5.0;
      A     #INT_xCrtPauseOrder;
      =     #OUT_xPauseOrder;
      A     L 5.0;
      A     #INT_xCrt13;
      =     #OUT_x13;
NETWORK
TITLE =
      A     #OUT_xLifeBitOk;
      A     #INT_xCrtStartStopPos;
      =     L 5.0;
      A     L 5.0;
      A     #IN_xOnline;
      =     L 5.1;
      A     L 5.1;
      A     #IN_SysTick;
      A(;
      L     #INT_iCntStartStopPos;
      L     10;
      <=I;
      );
      JNB   _00c;
      L     #INT_iCntStartStopPos;
      L     1;
      +I;
      T     #INT_iCntStartStopPos;
_00c: NOP   0;
      A     L 5.1;
      A(;
      L     #INT_iCntStartStopPos;
      L     10;
      >=I;
      );
      =     #OUT_xStartStopPos;
      A     L 5.0;
      NOT;
      JNB   _00d;
      L     0;
      T     #INT_iCntStartStopPos;
_00d: NOP   0;
NETWORK
TITLE =
      A     #OUT_xLifeBitOk;
      A     #INT_xReleaseOnline;
      =     #OUT_xReleaseOnline;
NETWORK
TITLE = set bits to master 1-7
      A     #ON;
      =     L 5.0;
      A     L 5.0;
      A     #IN_xFree;
      =     #INT_xStateFree;
      A     L 5.0;
      A     #IN_xOccupied;
      =     #INT_xStateOccupied;
      A     L 5.0;
      A     #IN_xLiftTop;
      =     #INT_xStateLiftTop;
      A     L 5.0;
      A     #IN_xOnline;
      =     #INT_xStateOnline;
      A     L 5.0;
      A     #IN_xReadyOnline;
      =     #INT_xStateReadyOnline;
      A     L 5.0;
      A     #IN_xError;
      =     #INT_xStateError;
      A     L 5.0;
      A     #IN_xMovingSource;
      =     #INT_xStateMovingSource;
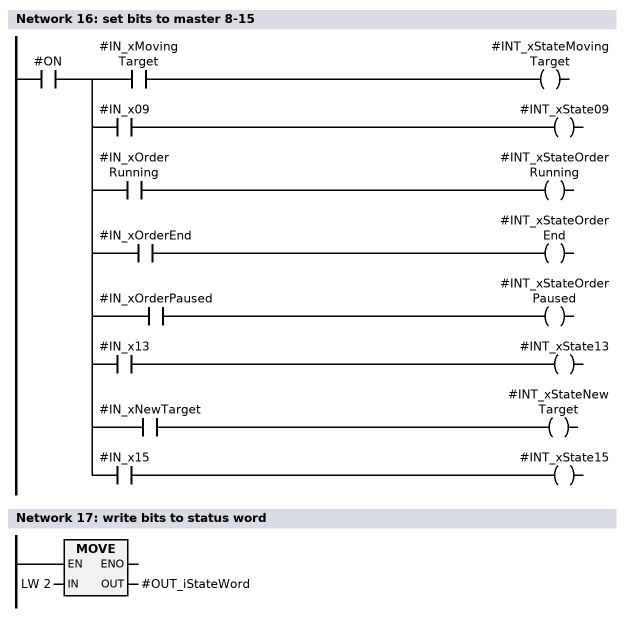
NETWORK
TITLE = set bits to master 8-15
      A     #ON;
      =     L 5.0;
      A     L 5.0;
      A     #IN_xMovingTarget;
      =     #INT_xStateMovingTarget;
      A     L 5.0;
      A     #IN_x09;
      =     #INT_xState09;
      A     L 5.0;
      A     #IN_xOrderRunning;
      =     #INT_xStateOrderRunning;
      A     L 5.0;
      A     #IN_xOrderEnd;
      =     #INT_xStateOrderEnd;
      A     L 5.0;
      A     #IN_xOrderPaused;
      =     #INT_xStateOrderPaused;
      A     L 5.0;
      A     #IN_x13;
      =     #INT_xState13;
      A     L 5.0;
      A     #IN_xNewTarget;
      =     #INT_xStateNewTarget;
      A     L 5.0;
      A     #IN_x15;
      =     #INT_xState15;
NETWORK
TITLE = write bits to status word
      L     LW 2;
      T     #OUT_iStateWord;
      NOP   0;
END_FUNCTION_BLOCK

FUNCTION_BLOCK "CheckEncoder"	// FB 21
TITLE = Check Encoder
VERSION : 0.1
VAR_INPUT
  ActualValue : DINT ;
  TurnMinus : BOOL ;
  TurnPlus : BOOL ;
  Reset : BOOL ;
  Clock_100ms : BOOL ;
  Clock_1s : BOOL ;
  minTurn : DINT ;
  maxTurn : DINT ;
  maxNotTurn : DINT ;
  fadeOut100ms : INT ;
END_VAR
VAR_OUTPUT
  Error : BOOL ;
  ErrorCode : INT ;
END_VAR
VAR
  lastValue : DINT ;
  actDiff : DINT ;
  p_Reset : BOOL ;
  p_Clock : BOOL ;
  p_Clock_1s : BOOL ;
  m_Error : BOOL ;
  timerTurn : INT ;
  timerNotTurn : INT ;
  m_ErrorCode : INT ;
  m_ErrorDiff : DINT ;
  timerCheck : INT ;
END_VAR
VAR_TEMP
  Clock : BOOL ;
  Turn : BOOL ;
  notTurn : BOOL ;
  Clock_1 : BOOL ;
END_VAR
BEGIN
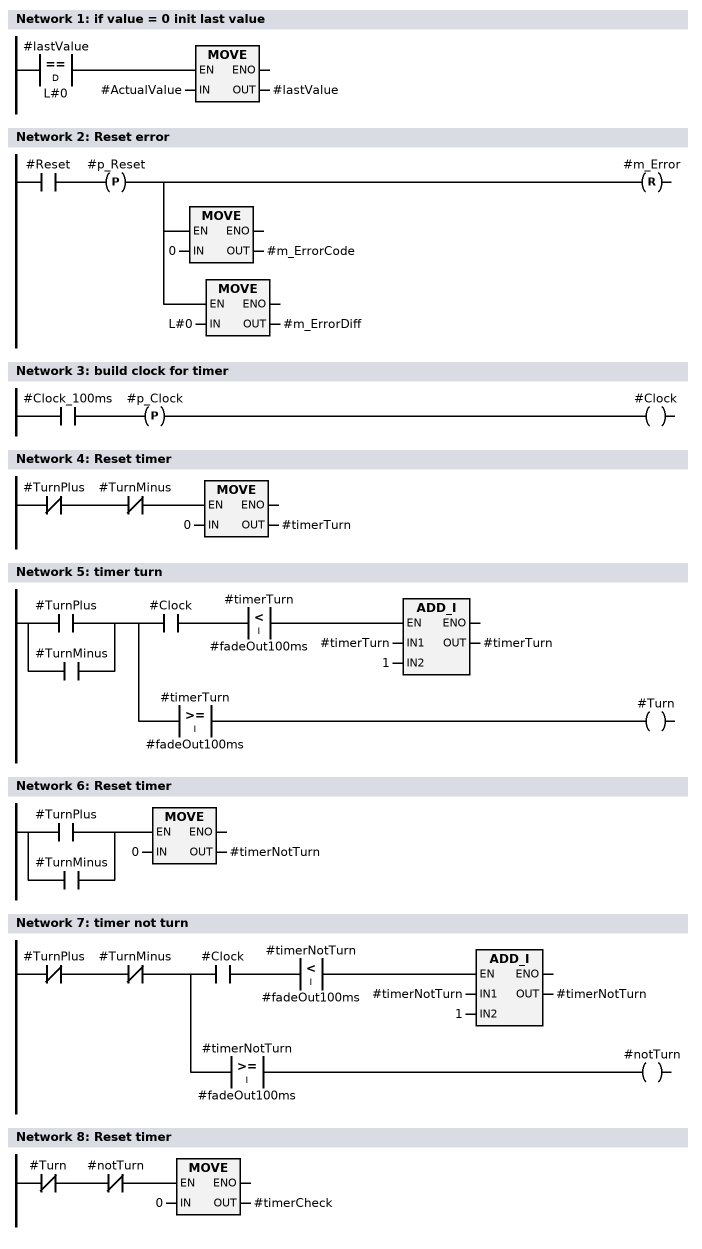
NETWORK
TITLE = if value = 0 init last value
      A(;
      L     #lastValue;
      L     L#0;
      ==D;
      );
      JNB   _001;
      L     #ActualValue;
      T     #lastValue;
_001: NOP   0;
NETWORK
TITLE = Reset error
      A     #Reset;
      FP    #p_Reset;
      =     L 1.0;
      A     L 1.0;
      BLD   102;
      R     #m_Error;
      A     L 1.0;
      JNB   _002;
      L     0;
      T     #m_ErrorCode;
_002: NOP   0;
      A     L 1.0;
      JNB   _003;
      L     L#0;
      T     #m_ErrorDiff;
_003: NOP   0;
NETWORK
TITLE = build clock for timer
      A     #Clock_100ms;
      FP    #p_Clock;
      =     #Clock;
NETWORK
TITLE = Reset timer
      AN    #TurnPlus;
      AN    #TurnMinus;
      JNB   _004;
      L     0;
      T     #timerTurn;
_004: NOP   0;
NETWORK
TITLE = timer turn
      O     #TurnPlus;
      O     #TurnMinus;
      =     L 1.0;
      A     L 1.0;
      A     #Clock;
      A(;
      L     #timerTurn;
      L     #fadeOut100ms;
      <I;
      );
      JNB   _005;
      L     #timerTurn;
      L     1;
      +I;
      T     #timerTurn;
_005: NOP   0;
      A     L 1.0;
      A(;
      L     #timerTurn;
      L     #fadeOut100ms;
      >=I;
      );
      =     #Turn;
NETWORK
TITLE = Reset timer
      A(;
      O     #TurnPlus;
      O     #TurnMinus;
      );
      JNB   _006;
      L     0;
      T     #timerNotTurn;
_006: NOP   0;
NETWORK
TITLE = timer not turn
      AN    #TurnPlus;
      AN    #TurnMinus;
      =     L 1.0;
      A     L 1.0;
      A     #Clock;
      A(;
      L     #timerNotTurn;
      L     #fadeOut100ms;
      <I;
      );
      JNB   _007;
      L     #timerNotTurn;
      L     1;
      +I;
      T     #timerNotTurn;
_007: NOP   0;
      A     L 1.0;
      A(;
      L     #timerNotTurn;
      L     #fadeOut100ms;
      >=I;
      );
      =     #notTurn;
NETWORK
TITLE = Reset timer
      AN    #Turn;
      AN    #notTurn;
      JNB   _008;
      L     0;
      T     #timerCheck;
_008: NOP   0;
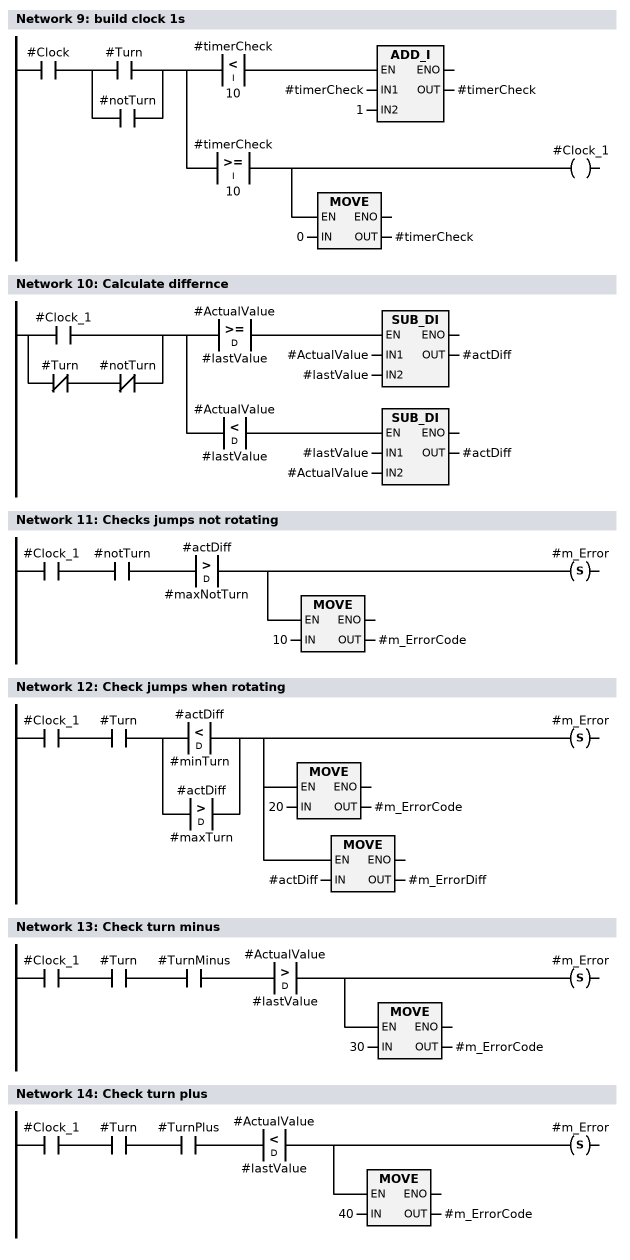
NETWORK
TITLE = build clock 1s
      A     #Clock;
      A(;
      O     #Turn;
      O     #notTurn;
      );
      =     L 1.0;
      A     L 1.0;
      A(;
      L     #timerCheck;
      L     10;
      <I;
      );
      JNB   _009;
      L     #timerCheck;
      L     1;
      +I;
      T     #timerCheck;
_009: NOP   0;
      A     L 1.0;
      A(;
      L     #timerCheck;
      L     10;
      >=I;
      );
      =     L 1.1;
      A     L 1.1;
      BLD   102;
      =     #Clock_1;
      A     L 1.1;
      JNB   _00a;
      L     0;
      T     #timerCheck;
_00a: NOP   0;
NETWORK
TITLE = Calculate differnce
      O     #Clock_1;
      O;
      AN    #Turn;
      AN    #notTurn;
      =     L 1.0;
      A     L 1.0;
      A(;
      L     #ActualValue;
      L     #lastValue;
      >=D;
      );
      JNB   _00b;
      L     #ActualValue;
      L     #lastValue;
      -D;
      T     #actDiff;
_00b: NOP   0;
      A     L 1.0;
      A(;
      L     #ActualValue;
      L     #lastValue;
      <D;
      );
      JNB   _00c;
      L     #lastValue;
      L     #ActualValue;
      -D;
      T     #actDiff;
_00c: NOP   0;
NETWORK
TITLE = Checks jumps not rotating
      A     #Clock_1;
      A     #notTurn;
      A(;
      L     #actDiff;
      L     #maxNotTurn;
      >D;
      );
      =     L 1.0;
      A     L 1.0;
      BLD   102;
      S     #m_Error;
      A     L 1.0;
      JNB   _00d;
      L     10;
      T     #m_ErrorCode;
_00d: NOP   0;
NETWORK
TITLE = Check jumps when rotating
      A     #Clock_1;
      A     #Turn;
      A(;
      O(;
      L     #actDiff;
      L     #minTurn;
      <D;
      );
      O(;
      L     #actDiff;
      L     #maxTurn;
      >D;
      );
      );
      =     L 1.0;
      A     L 1.0;
      BLD   102;
      S     #m_Error;
      A     L 1.0;
      JNB   _00e;
      L     20;
      T     #m_ErrorCode;
_00e: NOP   0;
      A     L 1.0;
      JNB   _00f;
      L     #actDiff;
      T     #m_ErrorDiff;
_00f: NOP   0;
NETWORK
TITLE = Check turn minus
      A     #Clock_1;
      A     #Turn;
      A     #TurnMinus;
      A(;
      L     #ActualValue;
      L     #lastValue;
      >D;
      );
      =     L 1.0;
      A     L 1.0;
      BLD   102;
      S     #m_Error;
      A     L 1.0;
      JNB   _010;
      L     30;
      T     #m_ErrorCode;
_010: NOP   0;
NETWORK
TITLE = Check turn plus
      A     #Clock_1;
      A     #Turn;
      A     #TurnPlus;
      A(;
      L     #ActualValue;
      L     #lastValue;
      <D;
      );
      =     L 1.0;
      A     L 1.0;
      BLD   102;
      S     #m_Error;
      A     L 1.0;
      JNB   _011;
      L     40;
      T     #m_ErrorCode;
_011: NOP   0;
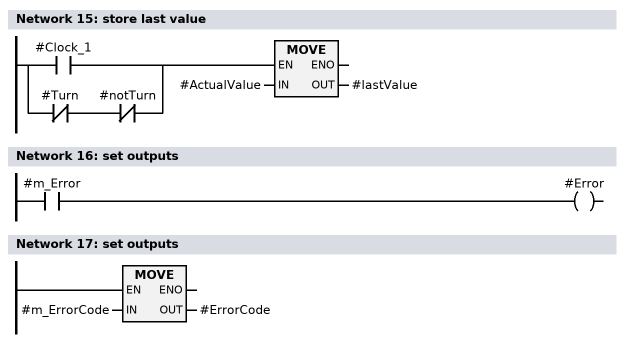
NETWORK
TITLE = store last value
      A(;
      O     #Clock_1;
      O;
      AN    #Turn;
      AN    #notTurn;
      );
      JNB   _012;
      L     #ActualValue;
      T     #lastValue;
_012: NOP   0;
NETWORK
TITLE = set outputs
      A     #m_Error;
      =     #Error;
NETWORK
TITLE = set outputs
      L     #m_ErrorCode;
      T     #ErrorCode;
      NOP   0;
END_FUNCTION_BLOCK

FUNCTION_BLOCK "GetCircumference"	// FB 22
//Ermittelt den Umfang aus einer Periode von Messungen
VERSION : 0.1
VAR_INPUT
  IN_Circum : INT ;
  IN_CntMax : INT ;
  IN_Takt : BOOL ;
  IN_Start : BOOL ;
  IN_Init : BOOL ;
END_VAR
VAR_OUTPUT
  OUT_End : BOOL ;
  OUT_OK : BOOL ;
END_VAR
VAR
  Value : ARRAY  [1 .. 10 ] OF DINT ;
  ChkVal : ARRAY  [1 .. 20 ] OF BOOL ;
  ChkValOK : ARRAY  [1 .. 20 ] OF BOOL ;
  Cnt : INT ;
  End : BOOL ;
  pFl1 : BOOL ;
  pFl2 : BOOL ;
END_VAR
VAR_TEMP
  Circum : DINT ;
  Cnt_Max : INT ;
  Wnd_Plu : DINT ;
  Wnd_Min : DINT ;
  Diff : DINT ;
  ON : BOOL ;
  Takt : BOOL ;
  Init : BOOL ;
  Mem : BOOL ;
  Chk : BOOL ;
END_VAR
BEGIN
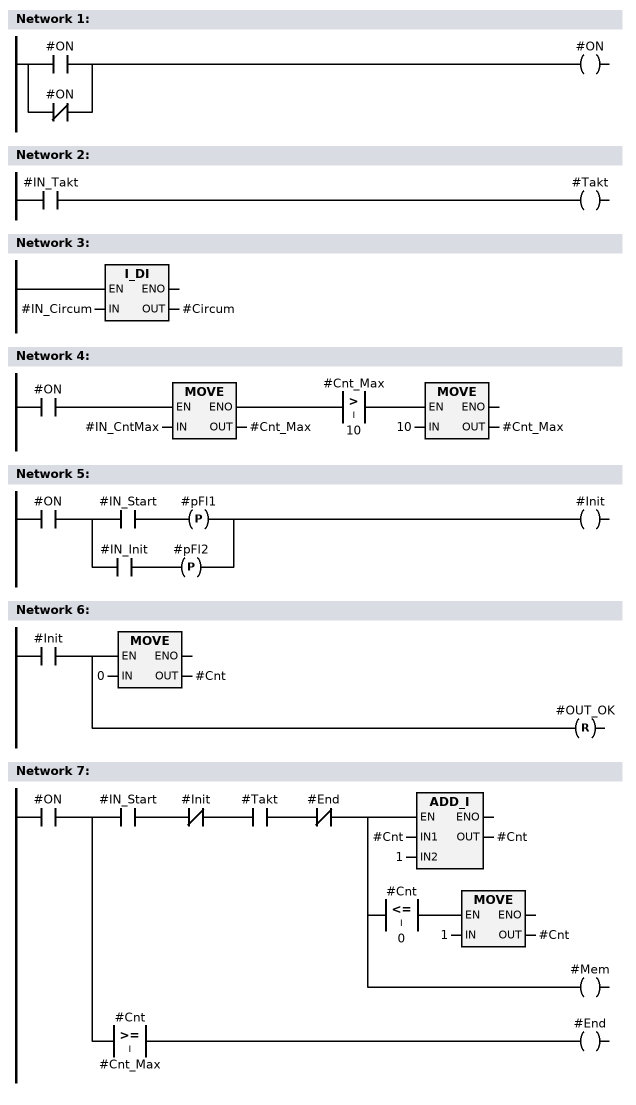
NETWORK
TITLE =
      O     #ON;
      ON    #ON;
      =     #ON;
NETWORK
TITLE =
      A     #IN_Takt;
      =     #Takt;
NETWORK
TITLE =
      L     #IN_Circum;
      ITD;
      T     #Circum;
      NOP   0;
NETWORK
TITLE =
      A(;
      A     #ON;
      JNB   _001;
      L     #IN_CntMax;
      T     #Cnt_Max;
      SET;
      SAVE;
      CLR;
_001: A     BR;
      );
      A(;
      L     #Cnt_Max;
      L     10;
      >I;
      );
      JNB   _002;
      L     10;
      T     #Cnt_Max;
_002: NOP   0;
NETWORK
TITLE =
      A     #ON;
      A(;
      O(;
      A     #IN_Start;
      BLD   100;
      FP    #pFl1;
      );
      O(;
      A     #IN_Init;
      BLD   100;
      FP    #pFl2;
      );
      );
      =     #Init;
NETWORK
TITLE =
      A     #Init;
      =     L 19.0;
      A     L 19.0;
      JNB   _003;
      L     0;
      T     #Cnt;
_003: NOP   0;
      A     L 19.0;
      BLD   102;
      R     #OUT_OK;
NETWORK
TITLE =
      A     #ON;
      =     L 19.0;
      A     L 19.0;
      A     #IN_Start;
      AN    #Init;
      A     #Takt;
      AN    #End;
      =     L 19.1;
      A     L 19.1;
      JNB   _004;
      L     #Cnt;
      L     1;
      +I;
      T     #Cnt;
_004: NOP   0;
      A     L 19.1;
      A(;
      L     #Cnt;
      L     0;
      <=I;
      );
      JNB   _005;
      L     1;
      T     #Cnt;
_005: NOP   0;
      A     L 19.1;
      BLD   102;
      =     #Mem;
      A     L 19.0;
      A(;
      L     #Cnt;
      L     #Cnt_Max;
      >=I;
      );
      =     #End;
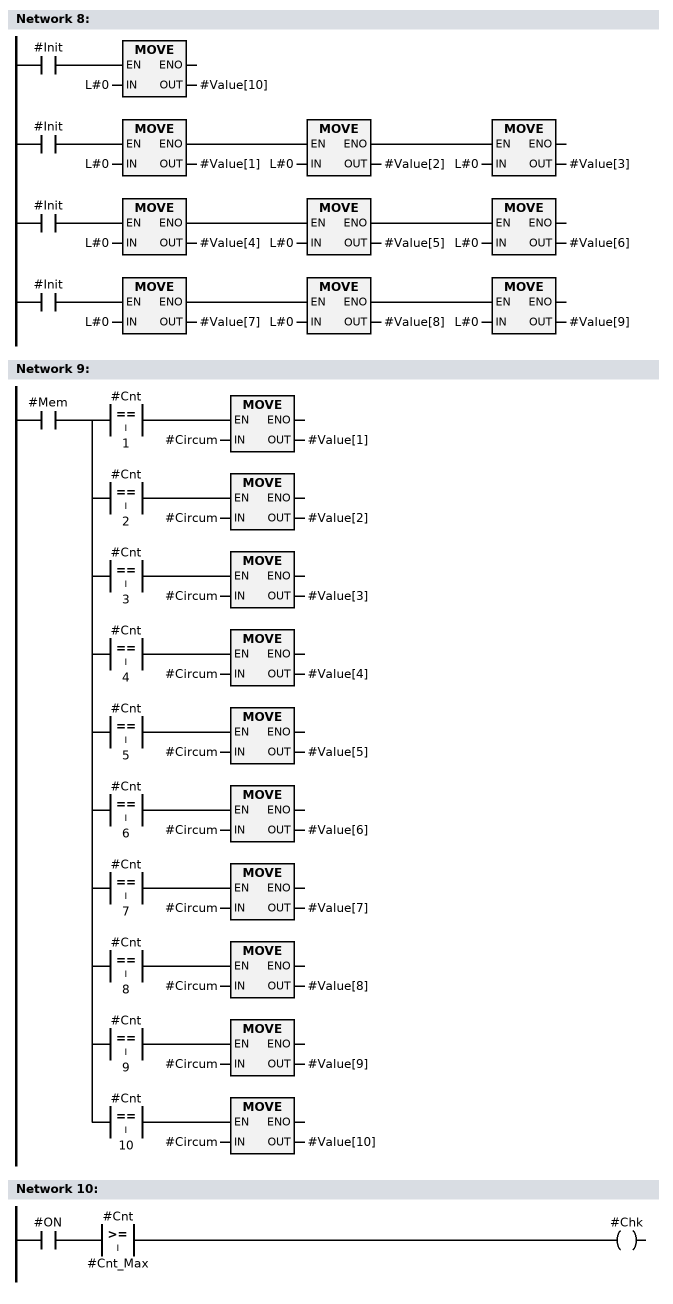
NETWORK
TITLE =
      A     #Init;
      =     L 19.0;
      A(;
      A(;
      A     L 19.0;
      JNB   _006;
      L     L#0;
      T     #Value[1];
      SET;
      SAVE;
      CLR;
_006: A     BR;
      );
      JNB   _007;
      L     L#0;
      T     #Value[2];
      SET;
      SAVE;
      CLR;
_007: A     BR;
      );
      JNB   _008;
      L     L#0;
      T     #Value[3];
_008: NOP   0;
      A(;
      A(;
      A     L 19.0;
      JNB   _009;
      L     L#0;
      T     #Value[4];
      SET;
      SAVE;
      CLR;
_009: A     BR;
      );
      JNB   _00a;
      L     L#0;
      T     #Value[5];
      SET;
      SAVE;
      CLR;
_00a: A     BR;
      );
      JNB   _00b;
      L     L#0;
      T     #Value[6];
_00b: NOP   0;
      A(;
      A(;
      A     L 19.0;
      JNB   _00c;
      L     L#0;
      T     #Value[7];
      SET;
      SAVE;
      CLR;
_00c: A     BR;
      );
      JNB   _00d;
      L     L#0;
      T     #Value[8];
      SET;
      SAVE;
      CLR;
_00d: A     BR;
      );
      JNB   _00e;
      L     L#0;
      T     #Value[9];
_00e: NOP   0;
      A     L 19.0;
      JNB   _00f;
      L     L#0;
      T     #Value[10];
_00f: NOP   0;
NETWORK
TITLE =
      A     #Mem;
      =     L 19.0;
      A     L 19.0;
      A(;
      L     #Cnt;
      L     1;
      ==I;
      );
      JNB   _010;
      L     #Circum;
      T     #Value[1];
_010: NOP   0;
      A     L 19.0;
      A(;
      L     #Cnt;
      L     2;
      ==I;
      );
      JNB   _011;
      L     #Circum;
      T     #Value[2];
_011: NOP   0;
      A     L 19.0;
      A(;
      L     #Cnt;
      L     3;
      ==I;
      );
      JNB   _012;
      L     #Circum;
      T     #Value[3];
_012: NOP   0;
      A     L 19.0;
      A(;
      L     #Cnt;
      L     4;
      ==I;
      );
      JNB   _013;
      L     #Circum;
      T     #Value[4];
_013: NOP   0;
      A     L 19.0;
      A(;
      L     #Cnt;
      L     5;
      ==I;
      );
      JNB   _014;
      L     #Circum;
      T     #Value[5];
_014: NOP   0;
      A     L 19.0;
      A(;
      L     #Cnt;
      L     6;
      ==I;
      );
      JNB   _015;
      L     #Circum;
      T     #Value[6];
_015: NOP   0;
      A     L 19.0;
      A(;
      L     #Cnt;
      L     7;
      ==I;
      );
      JNB   _016;
      L     #Circum;
      T     #Value[7];
_016: NOP   0;
      A     L 19.0;
      A(;
      L     #Cnt;
      L     8;
      ==I;
      );
      JNB   _017;
      L     #Circum;
      T     #Value[8];
_017: NOP   0;
      A     L 19.0;
      A(;
      L     #Cnt;
      L     9;
      ==I;
      );
      JNB   _018;
      L     #Circum;
      T     #Value[9];
_018: NOP   0;
      A     L 19.0;
      A(;
      L     #Cnt;
      L     10;
      ==I;
      );
      JNB   _019;
      L     #Circum;
      T     #Value[10];
_019: NOP   0;
NETWORK
TITLE =
      A     #ON;
      A(;
      L     #Cnt;
      L     #Cnt_Max;
      >=I;
      );
      =     #Chk;
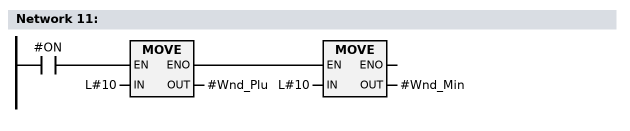
NETWORK
TITLE =
      A(;
      A     #ON;
      JNB   _01a;
      L     L#10;
      T     #Wnd_Plu;
      SET;
      SAVE;
      CLR;
_01a: A     BR;
      );
      JNB   _01b;
      L     L#10;
      T     #Wnd_Min;
_01b: NOP   0;
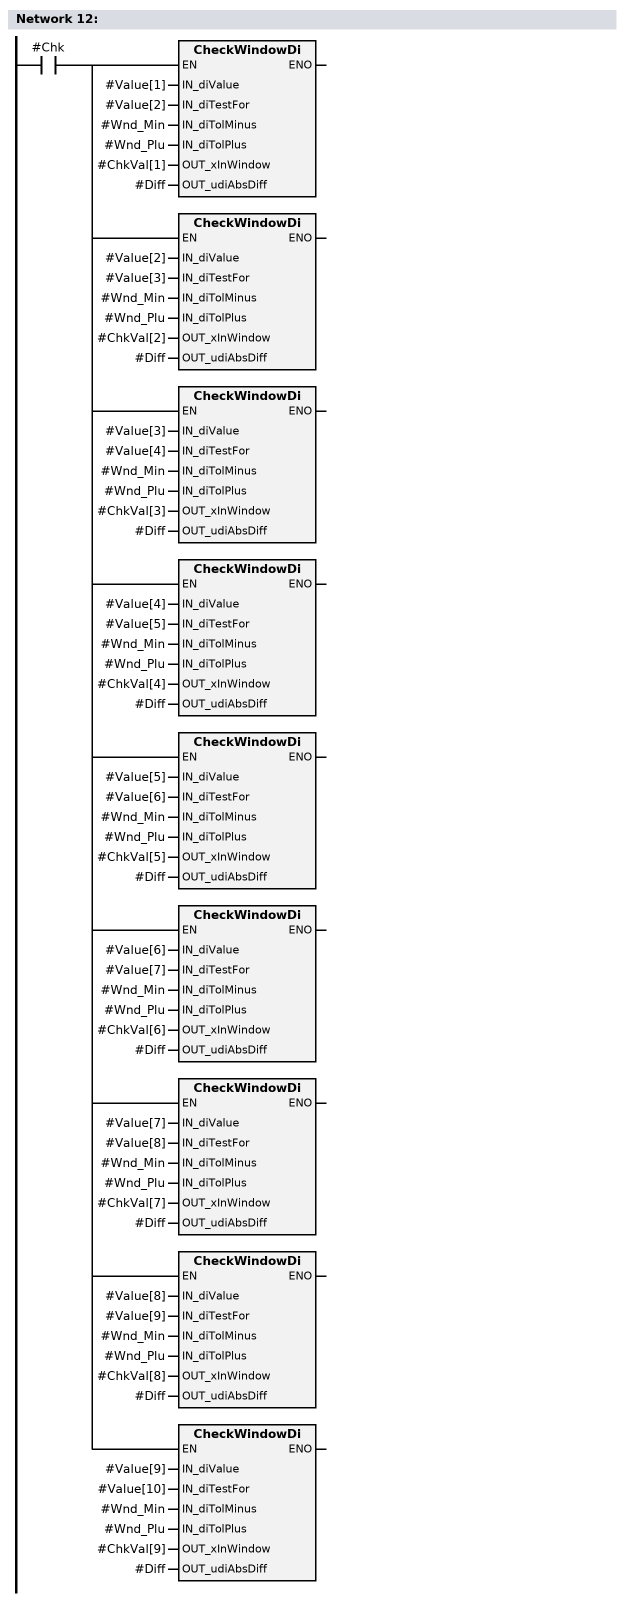
NETWORK
TITLE =
      A     #Chk;
      =     L 19.0;
      A     L 19.0;
      JNB   _01c;
      CALL  "CheckWindowDi" (
           IN_diValue               := #Value[1],
           IN_diTestFor             := #Value[2],
           IN_diTolMinus            := #Wnd_Min,
           IN_diTolPlus             := #Wnd_Plu,
           OUT_xInWindow            := #ChkVal[1],
           OUT_udiAbsDiff           := #Diff);
_01c: NOP   0;
      A     L 19.0;
      JNB   _01d;
      CALL  "CheckWindowDi" (
           IN_diValue               := #Value[2],
           IN_diTestFor             := #Value[3],
           IN_diTolMinus            := #Wnd_Min,
           IN_diTolPlus             := #Wnd_Plu,
           OUT_xInWindow            := #ChkVal[2],
           OUT_udiAbsDiff           := #Diff);
_01d: NOP   0;
      A     L 19.0;
      JNB   _01e;
      CALL  "CheckWindowDi" (
           IN_diValue               := #Value[3],
           IN_diTestFor             := #Value[4],
           IN_diTolMinus            := #Wnd_Min,
           IN_diTolPlus             := #Wnd_Plu,
           OUT_xInWindow            := #ChkVal[3],
           OUT_udiAbsDiff           := #Diff);
_01e: NOP   0;
      A     L 19.0;
      JNB   _01f;
      CALL  "CheckWindowDi" (
           IN_diValue               := #Value[4],
           IN_diTestFor             := #Value[5],
           IN_diTolMinus            := #Wnd_Min,
           IN_diTolPlus             := #Wnd_Plu,
           OUT_xInWindow            := #ChkVal[4],
           OUT_udiAbsDiff           := #Diff);
_01f: NOP   0;
      A     L 19.0;
      JNB   _020;
      CALL  "CheckWindowDi" (
           IN_diValue               := #Value[5],
           IN_diTestFor             := #Value[6],
           IN_diTolMinus            := #Wnd_Min,
           IN_diTolPlus             := #Wnd_Plu,
           OUT_xInWindow            := #ChkVal[5],
           OUT_udiAbsDiff           := #Diff);
_020: NOP   0;
      A     L 19.0;
      JNB   _021;
      CALL  "CheckWindowDi" (
           IN_diValue               := #Value[6],
           IN_diTestFor             := #Value[7],
           IN_diTolMinus            := #Wnd_Min,
           IN_diTolPlus             := #Wnd_Plu,
           OUT_xInWindow            := #ChkVal[6],
           OUT_udiAbsDiff           := #Diff);
_021: NOP   0;
      A     L 19.0;
      JNB   _022;
      CALL  "CheckWindowDi" (
           IN_diValue               := #Value[7],
           IN_diTestFor             := #Value[8],
           IN_diTolMinus            := #Wnd_Min,
           IN_diTolPlus             := #Wnd_Plu,
           OUT_xInWindow            := #ChkVal[7],
           OUT_udiAbsDiff           := #Diff);
_022: NOP   0;
      A     L 19.0;
      JNB   _023;
      CALL  "CheckWindowDi" (
           IN_diValue               := #Value[8],
           IN_diTestFor             := #Value[9],
           IN_diTolMinus            := #Wnd_Min,
           IN_diTolPlus             := #Wnd_Plu,
           OUT_xInWindow            := #ChkVal[8],
           OUT_udiAbsDiff           := #Diff);
_023: NOP   0;
      A     L 19.0;
      JNB   _024;
      CALL  "CheckWindowDi" (
           IN_diValue               := #Value[9],
           IN_diTestFor             := #Value[10],
           IN_diTolMinus            := #Wnd_Min,
           IN_diTolPlus             := #Wnd_Plu,
           OUT_xInWindow            := #ChkVal[9],
           OUT_udiAbsDiff           := #Diff);
_024: NOP   0;
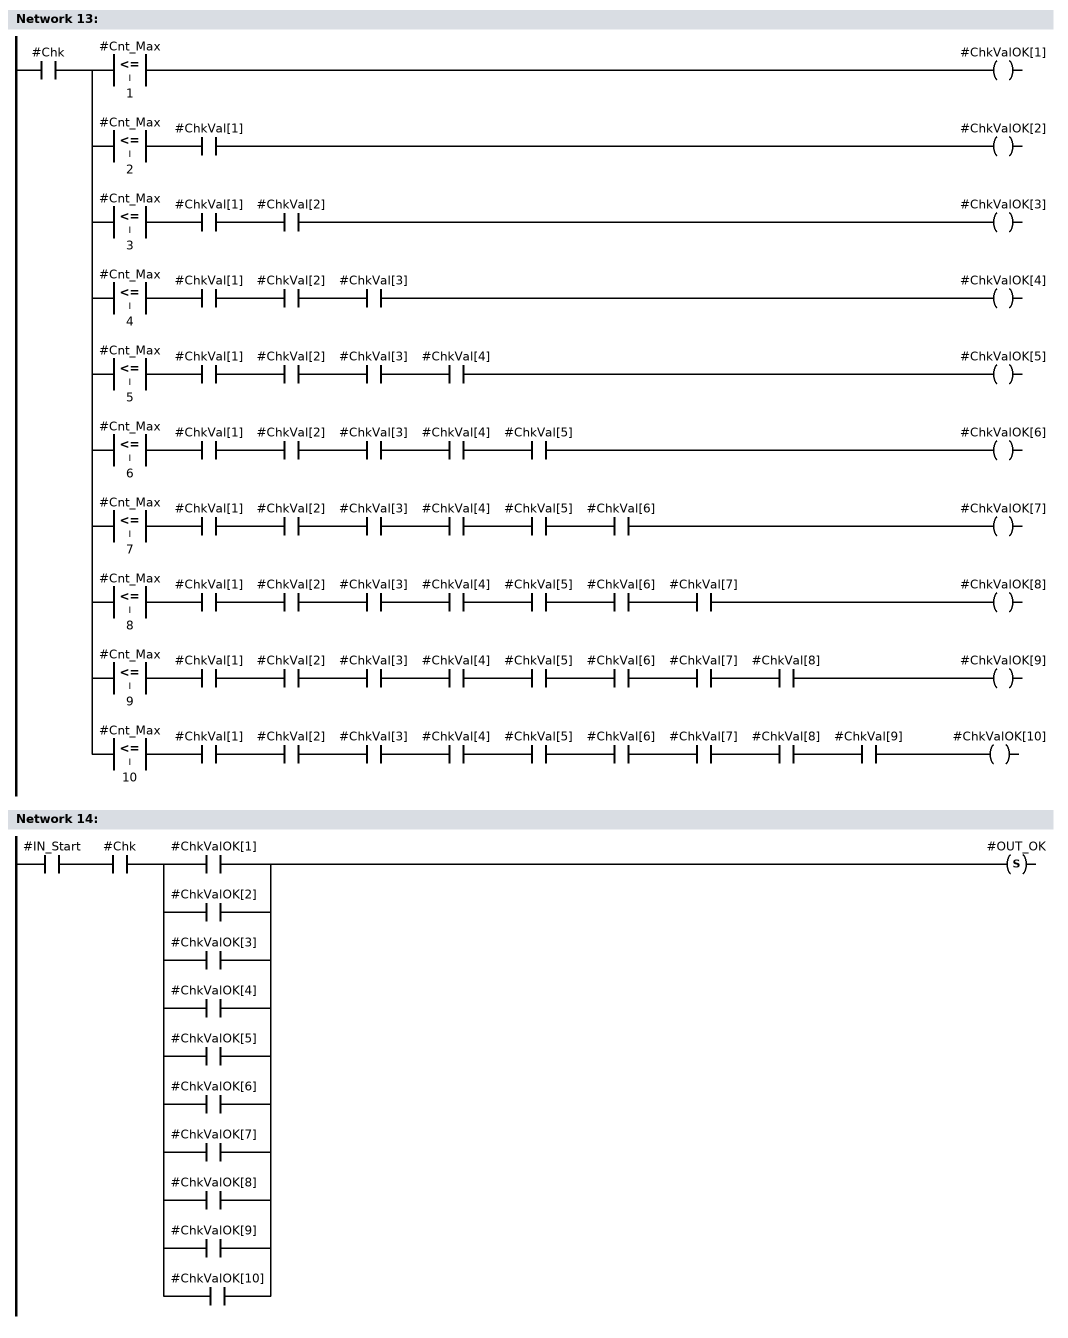
NETWORK
TITLE =
      A     #Chk;
      =     L 19.0;
      A     L 19.0;
      A(;
      L     #Cnt_Max;
      L     1;
      <=I;
      );
      =     #ChkValOK[1];
      A     L 19.0;
      A(;
      L     #Cnt_Max;
      L     2;
      <=I;
      );
      A     #ChkVal[1];
      =     #ChkValOK[2];
      A     L 19.0;
      A(;
      L     #Cnt_Max;
      L     3;
      <=I;
      );
      A     #ChkVal[1];
      A     #ChkVal[2];
      =     #ChkValOK[3];
      A     L 19.0;
      A(;
      L     #Cnt_Max;
      L     4;
      <=I;
      );
      A     #ChkVal[1];
      A     #ChkVal[2];
      A     #ChkVal[3];
      =     #ChkValOK[4];
      A     L 19.0;
      A(;
      L     #Cnt_Max;
      L     5;
      <=I;
      );
      A     #ChkVal[1];
      A     #ChkVal[2];
      A     #ChkVal[3];
      A     #ChkVal[4];
      =     #ChkValOK[5];
      A     L 19.0;
      A(;
      L     #Cnt_Max;
      L     6;
      <=I;
      );
      A     #ChkVal[1];
      A     #ChkVal[2];
      A     #ChkVal[3];
      A     #ChkVal[4];
      A     #ChkVal[5];
      =     #ChkValOK[6];
      A     L 19.0;
      A(;
      L     #Cnt_Max;
      L     7;
      <=I;
      );
      A     #ChkVal[1];
      A     #ChkVal[2];
      A     #ChkVal[3];
      A     #ChkVal[4];
      A     #ChkVal[5];
      A     #ChkVal[6];
      =     #ChkValOK[7];
      A     L 19.0;
      A(;
      L     #Cnt_Max;
      L     8;
      <=I;
      );
      A     #ChkVal[1];
      A     #ChkVal[2];
      A     #ChkVal[3];
      A     #ChkVal[4];
      A     #ChkVal[5];
      A     #ChkVal[6];
      A     #ChkVal[7];
      =     #ChkValOK[8];
      A     L 19.0;
      A(;
      L     #Cnt_Max;
      L     9;
      <=I;
      );
      A     #ChkVal[1];
      A     #ChkVal[2];
      A     #ChkVal[3];
      A     #ChkVal[4];
      A     #ChkVal[5];
      A     #ChkVal[6];
      A     #ChkVal[7];
      A     #ChkVal[8];
      =     #ChkValOK[9];
      A     L 19.0;
      A(;
      L     #Cnt_Max;
      L     10;
      <=I;
      );
      A     #ChkVal[1];
      A     #ChkVal[2];
      A     #ChkVal[3];
      A     #ChkVal[4];
      A     #ChkVal[5];
      A     #ChkVal[6];
      A     #ChkVal[7];
      A     #ChkVal[8];
      A     #ChkVal[9];
      =     #ChkValOK[10];
NETWORK
TITLE =
      A     #IN_Start;
      A     #Chk;
      A(;
      O     #ChkValOK[1];
      O     #ChkValOK[2];
      O     #ChkValOK[3];
      O     #ChkValOK[4];
      O     #ChkValOK[5];
      O     #ChkValOK[6];
      O     #ChkValOK[7];
      O     #ChkValOK[8];
      O     #ChkValOK[9];
      O     #ChkValOK[10];
      );
      S     #OUT_OK;
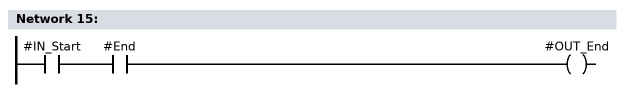
NETWORK
TITLE =
      A     #IN_Start;
      A     #End;
      =     #OUT_End;
END_FUNCTION_BLOCK

FUNCTION_BLOCK "WAGO_Analog_Input_4_20"	// FB 29
TITLE = Umfangsmessung mit lasersensor und WAGO-Analogeingabe 4-20mmA
//out_status_0 Messbereichsüberrschreitung
//out_status_1 + out_status_2 Messbereichsunterschreitung oder Leitungsbruch
//
VERSION : 0.1
VAR_INPUT
  in_enable : BOOL ;
  in_adresse : INT ;
  in_output_max : INT ;
  in_range_begin : INT ;
  in_range_end : INT ;
END_VAR
VAR_OUTPUT
  out_status_0 : BOOL ;
  out_status_1 : BOOL ;
  out_status_2 : BOOL ;
  i_distance : INT ;
END_VAR
VAR
  stat_referenz : REAL ;
END_VAR
VAR_TEMP
  tmp_status : STRUCT
   bit_0 : BOOL ;
   bit_1 : BOOL ;
   bit_2 : BOOL ;
   bit_3 : BOOL ;
   bit_4 : BOOL ;
   bit_5 : BOOL ;
   bit_6 : BOOL ;
   bit_7 : BOOL ;
  END_STRUCT ;
  tmp_adresse_1 : DWORD ;
  tmp_input : INT ;
  tmp_analog_val : INT ;
  tmp_messwert : REAL ;
  tmp_range_begin : REAL ;
  tmp_range_end : REAL ;
  tmp_diameter : REAL ;
  tmp_1 : REAL ;
  tmp_2 : REAL ;
  tmp_retval : WORD ;
  tmp_messwert_int : INT ;
END_VAR
BEGIN
NETWORK
TITLE = Initialisierung
      A     #in_enable;
      JC    M002;
      L     0;
      R     #out_status_0;
      R     #out_status_1;
      R     #out_status_2;
      T     #i_distance;
      JU    M001;
M002: NOP   0;
      L     #in_range_begin;
      DTR;
      T     #tmp_range_begin;
      L     #in_range_end;
      DTR;
      T     #tmp_range_end;
NETWORK
TITLE = Adresspointer
      L     #in_adresse;
      T     #tmp_adresse_1;
      SLD   3;
      T     #tmp_adresse_1;
NETWORK
TITLE = lese Eingangsdaten
      L     PIW [#tmp_adresse_1];
      T     #tmp_input;
NETWORK
TITLE = selektiere Analogwert
      L     #tmp_input;
      SRW   3;
      T     #tmp_analog_val;
NETWORK
TITLE = selektiere Statusbits
      L     #tmp_input;
      AW    W#16#7;
      T     #tmp_status;
      A     L 1.0;
      =     #out_status_0;
      A     L 1.1;
      =     #out_status_1;
      A     L 1.2;
      =     #out_status_2;
NETWORK
TITLE = scalierung
//Berechnung: Inc/mm = analogwert_max / Messbereich -> output_max / range_mm
//
      CALL  "SCALE_WAGO_AI" (
           IN                       := #tmp_analog_val,
           HI_LIM                   := #tmp_range_end,
           LO_LIM                   := #tmp_range_begin,
           BIPOLAR                  := FALSE,
           RET_VAL                  := #tmp_retval,
           OUT                      := #tmp_messwert);
NETWORK
TITLE = Roud to output
      L     #tmp_messwert;
      RND;
      T     #i_distance;
M001: NOP   0;
END_FUNCTION_BLOCK

// FB 37: know-how protected block, not included

// FB 63: know-how protected block, not included

// FB 64: know-how protected block, not included

// FB 65: know-how protected block, not included

// FB 66: know-how protected block, not included

FUNCTION_BLOCK "Safety_Position"	// FB 70
TITLE = Check safety positon
AUTHOR : Koenig
VERSION : 0.1
VAR_INPUT
  IN_Encoder_1_LO : INT ;	//Encoder 1 Low Word
  IN_Encoder_1_HI : INT ;	//Encoder 1 High Word
  IN_Encoder_2_LO : INT ;	//Encoder 2 Low Word
  IN_Encoder_2_HI : INT ;	//Encoder 2 High Word
  ReleaseFast : BOOL ;
  DiffSlow : INT ;
  DiffFast : INT ;
  Reset : BOOL ;
  Delay_CHK : TIME  := T#5S;
END_VAR
VAR_OUTPUT
  OUT_Difference_Lo : INT ;
  OUT_Difference_HI : INT ;
  Valid : BOOL ;
  Error_Diff : BOOL ;
END_VAR
VAR
  OFF : BOOL ;
  ON : BOOL ;
  delay : FB 186;
  checkDiff : BOOL ;
  err_Diff : BOOL ;
  delayTime : TIME  := T#1S;
  tmp_Difference_LO : INT ;
  tmp_Difference_HI : INT ;
  tmp_Encoder2_HI : INT ;
  tmp_lowerZero : BOOL ;
  tmp_ovBit_Sub1_LO : BOOL ;
  tmp_ovBit_Sub1_HI : BOOL ;
  tmp_ovBit_Mul1 : BOOL ;
  tmp_OFF : BOOL ;
  tmp_slow : BOOL ;
  chk_slow : BOOL ;
  t_slow : FB 185;
END_VAR
BEGIN
// body was compiled from another editor; compiled code not shown
END_FUNCTION_BLOCK

FUNCTION_BLOCK "Safety_Direction"	// FB 72
TITLE = Check direction
AUTHOR : Koenig
VERSION : 0.1
VAR_INPUT
  ActualPosition : INT ;
END_VAR
VAR_OUTPUT
  DirPlus : BOOL ;
  DirMinus : BOOL ;
  DirStop : BOOL ;
END_VAR
VAR
  LastValue : INT ;
  Change : BOOL ;
  DirectionPlus : BOOL ;
  DirectionMinus : BOOL ;
  TimeStop : TIME  := T#500MS;
  Stop : BOOL ;
  StartTimer : BOOL ;
  delay : FB 185;
END_VAR
BEGIN
// body was compiled from another editor; compiled code not shown
END_FUNCTION_BLOCK

FUNCTION_BLOCK "Safety_Speed"	// FB 73
AUTHOR : Koenig
VERSION : 0.1
VAR_INPUT
  ActPosition : INT ;
END_VAR
VAR
  LastPositon : INT ;
  Differnce : INT ;
  SpeedSecond : INT ;
  Speed : INT ;
  NoChange : BOOL ;
  error : BOOL ;
  TimeStop : TIME  := T#500MS;
  SpeedNull : BOOL ;
  Speed_1 : INT ;
  Speed_2 : INT ;
  Speed_3 : INT ;
  Calc : INT ;
  Result : INT ;
END_VAR
BEGIN
// body was compiled from another editor; compiled code not shown
END_FUNCTION_BLOCK

FUNCTION_BLOCK "Safety_SpeedCheck"	// FB 74
TITLE = Check safe speed speed
AUTHOR : Koenig
VERSION : 0.1
VAR_INPUT
  Reset : BOOL ;	//reset errors
  ReleaseFast : BOOL ;	//release fast speed
  CN_Stop : BOOL ;	//crane is not moving
  ActualSpeed : INT ;	//actual pseed in mm/s
  MaxSafeSpeed : INT ;	//max. safe speed in mm/s
  MaxSpeed : INT ;	//max. speed in mm/s
END_VAR
VAR_OUTPUT
  Error_SafeSpeed : BOOL ;
  Error_MaxSPeed : BOOL ;
END_VAR
VAR
  on : BOOL ;
  timeSafeSpeed : TIME  := T#4S;
  safeSpeed : BOOL ;
  nowCheck : BOOL ;
  DelayCheck : FB 185;
  err_SafeSpeed : BOOL ;
  err_Speed : BOOL ;
  err_OV : BOOL ;
  speed : INT ;
END_VAR
BEGIN
// body was compiled from another editor; compiled code not shown
END_FUNCTION_BLOCK

FUNCTION_BLOCK "Wago_Trolley"	// FB 81
TITLE = Check Hardware RBG Trolley / Lift
AUTHOR : Koenig
VERSION : 0.1
VAR_INPUT
  Reset : BOOL ;
END_VAR
VAR_OUTPUT
  HardwareOK : BOOL ;
END_VAR
VAR
  ON : BOOL ;
END_VAR
BEGIN
// body was compiled from another editor; compiled code not shown
END_FUNCTION_BLOCK

FUNCTION_BLOCK "F_Input_MAP"	// FB 91
TITLE = MAP safety input IOs (zones)
AUTHOR : Koenig
VERSION : 0.1
VAR
  ON : BOOL ;
  OFF : BOOL ;
  gblStopOK : BOOL ;
END_VAR
BEGIN
// body was compiled from another editor; compiled code not shown
END_FUNCTION_BLOCK

FUNCTION_BLOCK "ESTOP"	// FB 92
TITLE = ESTOP
AUTHOR : Koenig
VERSION : 0.1
VAR_INPUT
  Reset : BOOL ;
  Automatik : BOOL ;
END_VAR
VAR_OUTPUT
  ESTOP : BOOL ;
  ESTOP_DELAY : BOOL ;
END_VAR
VAR
  ON : BOOL ;
  Signal : BOOL ;
  M_ESTOP : BOOL ;
  Output : BOOL ;
  Q_Out_Delay : BOOL ;
END_VAR
BEGIN
// body was compiled from another editor; compiled code not shown
END_FUNCTION_BLOCK

FUNCTION_BLOCK "GetArea"	// FB 95
TITLE = Get zone (TR) for the position
VERSION : 0.1
VAR
  ON : BOOL ;
  Valid : BOOL ;
  BR_Value : INT ;
  TRTR_Dist : INT ;
  Calc : INT ;
  TR_rel_Value : INT ;
  TR_Value : INT ;
END_VAR
BEGIN
// body was compiled from another editor; compiled code not shown
END_FUNCTION_BLOCK

// FB 101: know-how protected block, not included

FUNCTION_BLOCK "MODBUSPN"	// FB 102
TITLE = MODBUSPN
AUTHOR : SIEMENS
FAMILY : COMM
NAME : MODBUSPN
VERSION : 3.4
VAR_INPUT
  ID : WORD ;
  DB_PARAM : BLOCK_DB ;
  RECV_TIME : TIME ;
  CONN_TIME : TIME ;
  KEEP_ALIVE : TIME ;
  ENQ_ENR : BOOL ;
  DISCONNECT : BOOL ;
  REG_KEY : STRING  [17 ] := '                 ';
END_VAR
VAR_OUTPUT
  LICENSED : BOOL ;
  BUSY : BOOL ;
  CONN_ESTABLISHED : BOOL ;
  DONE_NDR : BOOL ;
  ERROR : BOOL ;
  STATUS_MODBUS : WORD ;
  STATUS_CONN : WORD ;
  STATUS_FUNC : STRING  [8 ];
  IDENT_CODE : STRING  [18 ];
END_VAR
VAR_IN_OUT
  UNIT : BYTE ;
  DATA_TYPE : BYTE ;
  START_ADDRESS : WORD ;
  LENGTH : WORD ;
  TI : WORD ;
  WRITE_READ : BOOL ;
END_VAR
VAR
  TEST_DB : STRUCT
   RET_WERT : INT ;
   LENGTH : WORD ;
   WRITE_PROTECT : BOOL ;
  END_STRUCT ;
  MOD_CLI : FB 104;
  MOD_SERV : FB 105;
  TON : SFB 4;
  sID : WORD ;
  sWDB_PARAM : WORD ;
  sSTATUS_TEMP : WORD ;
  sSTATUS_TIMER : WORD ;
  sSTATUS_FUNC : STRING  [8 ];
  sSTATUS_CODE : STRING  [17 ];
  sOFFSET_PARAM : DINT ;
  sCONN_TIME : TIME ;
  sPTR_SEND_BUFFER : DINT ;
  sPTR_RECV1_BUFFER : DINT ;
  sPTR_RECV2_BUFFER : DINT ;
  sSERVER_CLIENT : BOOL ;
  sSINGLE_WRITE : BOOL ;
  sC_AT_STARTUP : BOOL ;
  sANLAUF_FEHLER : BOOL ;
  sID_GEFUNDEN : BOOL ;
  sAREA_VALID : ARRAY  [1 .. 8 ] OF BOOL ;
  sAREA_1 : ARRAY  [1 .. 2 ] OF CHAR  := 'M', 'O';
  sAREA_2 : ARRAY  [1 .. 4 ] OF CHAR  := 'D', 'B', 'U', 'S';
  tStart_x : DINT ;
  tEnd_x : DINT ;
  tStart_y : DINT ;
  tEnd_y : DINT ;
  tDBLength_650 : INT ;
  tDbNr : WORD ;
  i : INT ;
  j : INT ;
  pos : INT ;
  sDataType : WORD ;
  snd_time : BYTE ;
  rcv_time : BYTE ;
  sACODE : ARRAY  [0 .. 17 ] OF BYTE ;
  RD_SINFO : STRUCT
   RET_WERT : INT ;
   TOP_SI : STRUCT
    EV_CLASS : BYTE ;
    EV_NUM : BYTE ;
    PRIORITY : BYTE ;
    NUM : BYTE ;
    TYP2_3 : BYTE ;
    TYP1 : BYTE ;
    ZI1 : WORD ;
    ZI2_3 : DWORD ;
   END_STRUCT ;
   START_UP_SI : STRUCT
    EV_CLASS : BYTE ;
    EV_NUM : BYTE ;
    PRIORITY : BYTE ;
    NUM : BYTE ;
    TYP2_3 : BYTE ;
    TYP1 : BYTE ;
    ZI1 : WORD ;
    ZI2_3 : DWORD ;
   END_STRUCT ;
  END_STRUCT ;
  RDSYSST : STRUCT
   RET_WERT : INT ;
   REQ : BOOL ;
   BUSY : BOOL ;
   SZL_HEADER : STRUCT
    LENTHDR : WORD ;
    N_DR : WORD ;
   END_STRUCT ;
   SZL_11C_5 : STRUCT
    index : WORD ;
    serialn : ARRAY  [0 .. 23 ] OF CHAR ;
    res : ARRAY  [1 .. 4 ] OF WORD ;
   END_STRUCT ;
  END_STRUCT ;
  sHoldingRegisterState : ARRAY  [0 .. 24 ] OF BYTE ;
END_VAR
VAR_TEMP
  tSProductID : STRING  [19 ];
  tALicenseKey : ARRAY  [0 .. 17 ] OF BYTE ;
END_VAR
BEGIN
NETWORK
TITLE = SCL network
//compiled by SCL compiler version:  SCLCOMP K05.03.05.00_01.03.00.01 release
// (network holds code this reader does not know; not shown)
END_FUNCTION_BLOCK

FUNCTION_BLOCK "TCP_COMM"	// FB 103
TITLE = TCP_COMM
AUTHOR : SIEMENS
FAMILY : COMM
NAME : TCP_COMM
VERSION : 3.0
VAR_INPUT
  ID : WORD ;
  DATA_TRANSFER : BOOL ;
  SEND_RCV : BOOL ;
  CONNECT_DISCONNECT : BOOL ;
  LENGTH : INT ;
  MONITOR : TIME ;
  KEEP_ALIVE : BOOL ;
  ANLAUF : BOOL ;
END_VAR
VAR_OUTPUT
  CONN_ESTABLISHED : BOOL ;
  BUSY : BOOL ;
  DONE : BOOL ;
  ERROR : BOOL ;
  STATUS : WORD ;
  STATUS_FUNC : STRING  [8 ];
END_VAR
VAR_IN_OUT
  ENQ : BOOL ;
  UDT_CONN : ANY ;
  DATA : ANY ;
END_VAR
VAR
  TCON : FB 65;
  TSEND : FB 63;
  TRCV : FB 64;
  TDISCON : FB 66;
  TON : SFB 4;
  TDISCON_MONITORING : TIME ;
  MONITOR_TIME : TIME ;
  i : INT ;
  MONITOR_active : BOOL ;
  MONITOR_OUT : BOOL ;
  TCON_Req : BOOL ;
  TSEND_Req : BOOL ;
  TRCV_Req : BOOL ;
  TDISCON_Req : BOOL ;
  TCON_Busy : BOOL ;
  TSEND_Busy : BOOL ;
  TRCV_Busy : BOOL ;
  TDISCON_Busy : BOOL ;
  ENQ_Save : BOOL ;
  Req : BOOL ;
  OrderErrorDiscon : BOOL ;
  Order_new_TCON : BOOL ;
  Order_again_TCON : BOOL ;
  Order_immed_TSEND : BOOL ;
  Order_immed_TDCON : BOOL ;
END_VAR
BEGIN
// body was compiled from an SCL source; compiled code not shown
END_FUNCTION_BLOCK

FUNCTION_BLOCK "MOD_CLI"	// FB 104
TITLE = MOD_CLI
AUTHOR : SIEMENS
FAMILY : COMM
NAME : MOD_CLI
VERSION : 1.5
VAR_INPUT
  ID : WORD ;
  DB_PARAM : BLOCK_DB ;
  WDB_PARAM : WORD ;
  RECV_TIME : TIME ;
  CONN_TIME : TIME ;
  sC_AT_STARTUP : BOOL ;
  ENQ_ENR : BOOL ;
  DISCONNECT : BOOL ;
  SERVER_CLIENT : BOOL ;
  ANLAUF : BOOL ;
  SINGLE_WRITE : BOOL ;
  OFFSET_PARAM : DINT ;
  PTR_SEND_BUFFER : DINT ;
  PTR_RECV1_BUFFER : DINT ;
  PTR_RECV2_BUFFER : DINT ;
  sAREA_VALID : ARRAY  [1 .. 8 ] OF BOOL ;
  SRCBLK_Struct : STRUCT
   ANY_id : WORD ;
   Length : WORD ;
   DB_Number : WORD ;
   Byte_Pointer : DWORD ;
  END_STRUCT ;
  TCON_Struct : STRUCT
   ANY_id : WORD ;
   Length : WORD ;
   DB_Number : WORD ;
   Byte_Pointer : DWORD ;
  END_STRUCT ;
  DSTBLK_Struct : STRUCT
   ANY_id : WORD ;
   Length : WORD ;
   DB_Number : WORD ;
   Byte_Pointer : DWORD ;
  END_STRUCT ;
END_VAR
VAR_OUTPUT
  BUSY : BOOL ;
  CONN_ESTABLISHED : BOOL ;
  ERROR : BOOL ;
  STATUS_MODBUS : WORD ;
  STATUS_CONN : WORD ;
  STATUS_FUNC : STRING  [8 ];
END_VAR
VAR_IN_OUT
  UNIT : BYTE ;
  DATA_TYPE : BYTE ;
  START_ADDRESS : WORD ;
  LENGTH : WORD ;
  TI : WORD ;
  WRITE_READ : BOOL ;
  DONE_NDR : BOOL ;
END_VAR
VAR
  TEST_DB : STRUCT
   RET_WERT : INT ;
   LENGTH : WORD ;
   WRITE_PROTECT : BOOL ;
  END_STRUCT ;
  STATE : STRUCT
   AUFTRAG_LAEUFT : BOOL ;
   SEND : BOOL ;
   RECV1 : BOOL ;
   RECV2 : BOOL ;
   EXCEPT : BOOL ;
   CON : BOOL ;
   SENDEDATEN_DA : BOOL ;
   WARTEN_AUF_VERB : BOOL ;
  END_STRUCT ;
  TCP_COMM : FB 103;
  sUNIT : BYTE ;
  sFUNC_CODE : BYTE ;
  sDATA_TYPE : BYTE ;
  sVariable_1 : BYTE ;
  sCoil_On_Off : BYTE ;
  sVariable_2 : BYTE ;
  sShift_left : BYTE ;
  sShift_rigth : BYTE ;
  sDATEN_DB : WORD ;
  sNUMBER_OF_VALUES : INT ;
  sDATEN_START : DINT ;
  sSTART_ADDRESS : DINT ;
  sTI : WORD ;
  sIDB_Nr : WORD ;
  sLEN_RECV2 : INT ;
  sSTATUS_TEMP : WORD ;
  sRECV_TIME : TIME ;
  sClient_Req_senden : BOOL ;
  sSenden : BOOL ;
  sDISCON : BOOL ;
  sWRITE_READ : BOOL ;
  sLAST_ENQ_ENR : BOOL ;
  sFirstBit_Grenze0 : BOOL ;
  sLength_groesser_8 : BOOL ;
  slength_Multiple_8 : BOOL ;
  sZustaende_loeschen : BOOL ;
  i : INT ;
  j : INT ;
  sBLKMOV_RET_VAL : INT ;
  sOFFSET_DATEN : DINT ;
  sExc_BytCnt_StaAdr : DINT ;
  sStart_x : DINT ;
  sEnd_x : DINT ;
  sFirst_Bit : INT ;
  sFirst_Byte : INT ;
  sLast_Bit : INT ;
  sLast_Byte : INT ;
  sByteCount_Bit : INT ;
END_VAR
BEGIN
// body was compiled from an SCL source; compiled code not shown
END_FUNCTION_BLOCK

FUNCTION_BLOCK "MOD_SERV"	// FB 105
TITLE = MOD_SERV
AUTHOR : SIEMENS
FAMILY : COMM
NAME : MOD_SERV
VERSION : 1.3
VAR_INPUT
  ID : WORD ;
  DB_PARAM : BLOCK_DB ;
  WDB_PARAM : WORD ;
  RECV_TIME : TIME ;
  CONN_TIME : TIME ;
  sC_AT_STARTUP : BOOL ;
  ENQ_ENR : BOOL ;
  DISCONNECT : BOOL ;
  SERVER_CLIENT : BOOL ;
  ANLAUF : BOOL ;
  OFFSET_PARAM : DINT ;
  PTR_SEND_BUFFER : DINT ;
  PTR_RECV1_BUFFER : DINT ;
  PTR_RECV2_BUFFER : DINT ;
  SRCBLK_Struct : STRUCT
   ANY_id : WORD ;
   Length : WORD ;
   DB_Number : WORD ;
   Byte_Pointer : DWORD ;
  END_STRUCT ;
  DSTBLK_Struct : STRUCT
   ANY_id : WORD ;
   Length : WORD ;
   DB_Number : WORD ;
   Byte_Pointer : DWORD ;
  END_STRUCT ;
END_VAR
VAR_OUTPUT
  UNIT : BYTE ;
  DATA_TYPE : BYTE ;
  START_ADDRESS : WORD ;
  LENGTH : WORD ;
  TI : WORD ;
  WRITE_READ : BOOL ;
  DONE_NDR : BOOL ;
  BUSY : BOOL ;
  CONN_ESTABLISHED : BOOL ;
  ERROR : BOOL ;
  STATUS_MODBUS : WORD ;
  STATUS_CONN : WORD ;
  STATUS_FUNC : STRING  [8 ];
END_VAR
VAR
  TEST_DB : STRUCT
   RET_WERT : INT ;
   LENGTH : WORD ;
   WRITE_PROTECT : BOOL ;
  END_STRUCT ;
  STATE : STRUCT
   AUFTRAG_LAEUFT : BOOL ;
   SEND : BOOL ;
   RECV1 : BOOL ;
   RECV2 : BOOL ;
   EXCEPT : BOOL ;
   CON : BOOL ;
   SENDEDATEN_DA : BOOL ;
   WARTEN_AUF_VERB : BOOL ;
  END_STRUCT ;
  TCP_COMM : FB 103;
  sCoil_On_Off : BYTE ;
  sEXCEPTION_CODE : BYTE ;
  sFUNC_CODE : BYTE ;
  sDATA_TYPE : BYTE ;
  sUnit : BYTE ;
  sVariable_1 : BYTE ;
  sVariable_2 : BYTE ;
  sShift_left : BYTE ;
  sShift_rigth : BYTE ;
  sDISCON : BOOL ;
  sWRITE_READ : BOOL ;
  sZustaende_loeschen : BOOL ;
  sSend_Aufrufen : BOOL ;
  sFirstBit_Grenze0 : BOOL ;
  sLength_groesser_8 : BOOL ;
  slength_Multiple_8 : BOOL ;
  sDATEN_DB : WORD ;
  sIDB_Nr : WORD ;
  sTI : WORD ;
  sDATEN_START : DINT ;
  sSTART_ADDRESS : DINT ;
  sNUMBER_OF_VALUES : INT ;
  sLEN_RECV2 : INT ;
  sByteCount_Bit : INT ;
  sCONN_TIME : TIME ;
  sRECV_TIME : TIME ;
  i : INT ;
  j : INT ;
  sBLKMOV_RET_VAL : INT ;
  sOFFSET_DATEN : DINT ;
  sFirst_Bit : INT ;
  sFirst_Byte : INT ;
  sLast_Bit : INT ;
  sLast_Byte : INT ;
  sSTATUS_FUNC : STRING  [8 ];
END_VAR
BEGIN
// body was compiled from an SCL source; compiled code not shown
END_FUNCTION_BLOCK

// FB 126: know-how protected block, not included

// FB 127: know-how protected block, not included

// FB 185: know-how protected block, not included

// FB 186: know-how protected block, not included

FUNCTION_BLOCK "CopyHookDBs"	// FB 190
VERSION : 0.1
VAR_INPUT
  DB_Source1 : INT ;
  DB_Target1 : INT ;
  DB_Source2 : INT ;
  DB_Target2 : INT ;
  Start : BOOL ;
END_VAR
VAR_OUTPUT
  OUT_RetVal : INT ;
END_VAR
VAR_IN_OUT
  IO_Busy : BOOL ;
END_VAR
VAR
  T_Delay : SFB 4;
  T_ChkRuntime : SFB 4;
  ReadDBL : FB 192;
  INT_DB_Source1 : INT ;
  INT_DB_Target1 : INT ;
  INT_DB_Source2 : INT ;
  INT_DB_Target2 : INT ;
  INT_DB_Length : INT ;
  INT_Step : INT ;
  INT_RetVal1 : INT ;
  INT_RetVal2 : INT ;
  INT_RetVal3 : INT ;
  INT_StepDel : BOOL ;
  Edge1 : BOOL ;
  Edge2 : BOOL ;
  Edge3 : BOOL ;
  Edge4 : BOOL ;
  INT_Busy : BOOL ;
  Edge_Start : BOOL ;
  ReadyDBL : BOOL ;
  ready1 : BOOL ;
  ready2 : BOOL ;
  DB1_finished : BOOL ;
  DB2_finished : BOOL ;
  tmp_StartDBL : BOOL ;
  tmp_DB_Source : INT ;
  tmp_DB_Target : INT ;
  tmp_DB_Length : INT ;
END_VAR
VAR_TEMP
  tmp_RetVal : INT ;
  tmp_RetVal_Src : INT ;
  tmp_Test1 : INT ;
  tmp_Test2 : INT ;
  tmp_DB_Src_Word : WORD ;
  tmp_DB_Src_Length : WORD ;
  tmp_DB_Src_Protect : BOOL ;
  tmp_test : INT ;
END_VAR
BEGIN
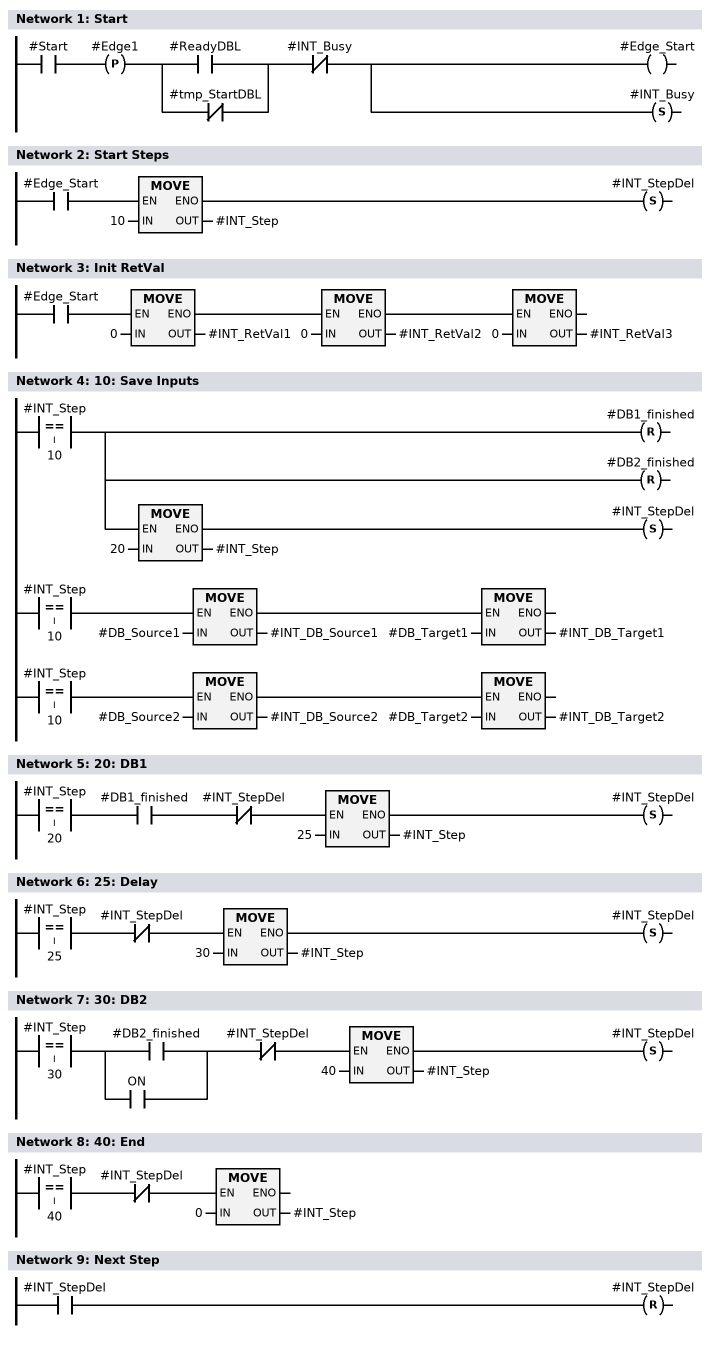
NETWORK
TITLE = Start
      A     #Start;
      FP    #Edge1;
      A(;
      O     #ReadyDBL;
      ON    #tmp_StartDBL;
      );
      AN    #INT_Busy;
      =     #Edge_Start;
      S     #INT_Busy;
NETWORK
TITLE = Start Steps
      A     #Edge_Start;
      JNB   _001;
      L     10;
      T     #INT_Step;
      SET;
      SAVE;
      CLR;
_001: A     BR;
      S     #INT_StepDel;
NETWORK
TITLE = Init RetVal
      A(;
      A(;
      A     #Edge_Start;
      JNB   _002;
      L     0;
      T     #INT_RetVal1;
      SET;
      SAVE;
      CLR;
_002: A     BR;
      );
      JNB   _003;
      L     0;
      T     #INT_RetVal2;
      SET;
      SAVE;
      CLR;
_003: A     BR;
      );
      JNB   _004;
      L     0;
      T     #INT_RetVal3;
_004: NOP   0;
NETWORK
TITLE = 10: Save Inputs
      L     #INT_Step;
      L     10;
      ==I;
      =     L 16.0;
      A(;
      A     L 16.0;
      JNB   _005;
      L     #DB_Source1;
      T     #INT_DB_Source1;
      SET;
      SAVE;
      CLR;
_005: A     BR;
      );
      JNB   _006;
      L     #DB_Target1;
      T     #INT_DB_Target1;
_006: NOP   0;
      A(;
      A     L 16.0;
      JNB   _007;
      L     #DB_Source2;
      T     #INT_DB_Source2;
      SET;
      SAVE;
      CLR;
_007: A     BR;
      );
      JNB   _008;
      L     #DB_Target2;
      T     #INT_DB_Target2;
_008: NOP   0;
      A     L 16.0;
      BLD   102;
      R     #DB1_finished;
      A     L 16.0;
      BLD   102;
      R     #DB2_finished;
      A     L 16.0;
      JNB   _009;
      L     20;
      T     #INT_Step;
      SET;
      SAVE;
      CLR;
_009: A     BR;
      S     #INT_StepDel;
NETWORK
TITLE = 20: DB1
      A(;
      L     #INT_Step;
      L     20;
      ==I;
      );
      A     #DB1_finished;
      AN    #INT_StepDel;
      JNB   _00a;
      L     25;
      T     #INT_Step;
      SET;
      SAVE;
      CLR;
_00a: A     BR;
      S     #INT_StepDel;
NETWORK
TITLE = 25: Delay
      A(;
      L     #INT_Step;
      L     25;
      ==I;
      );
      AN    #INT_StepDel;
      JNB   _00b;
      L     30;
      T     #INT_Step;
      SET;
      SAVE;
      CLR;
_00b: A     BR;
      S     #INT_StepDel;
NETWORK
TITLE = 30: DB2
      A(;
      L     #INT_Step;
      L     30;
      ==I;
      );
      A(;
      O     #DB2_finished;
      O     "ON";
      );
      AN    #INT_StepDel;
      JNB   _00c;
      L     40;
      T     #INT_Step;
      SET;
      SAVE;
      CLR;
_00c: A     BR;
      S     #INT_StepDel;
NETWORK
TITLE = 40: End
      A(;
      L     #INT_Step;
      L     40;
      ==I;
      );
      AN    #INT_StepDel;
      JNB   _00d;
      L     0;
      T     #INT_Step;
_00d: NOP   0;
NETWORK
TITLE = Next Step
      A     #INT_StepDel;
      R     #INT_StepDel;
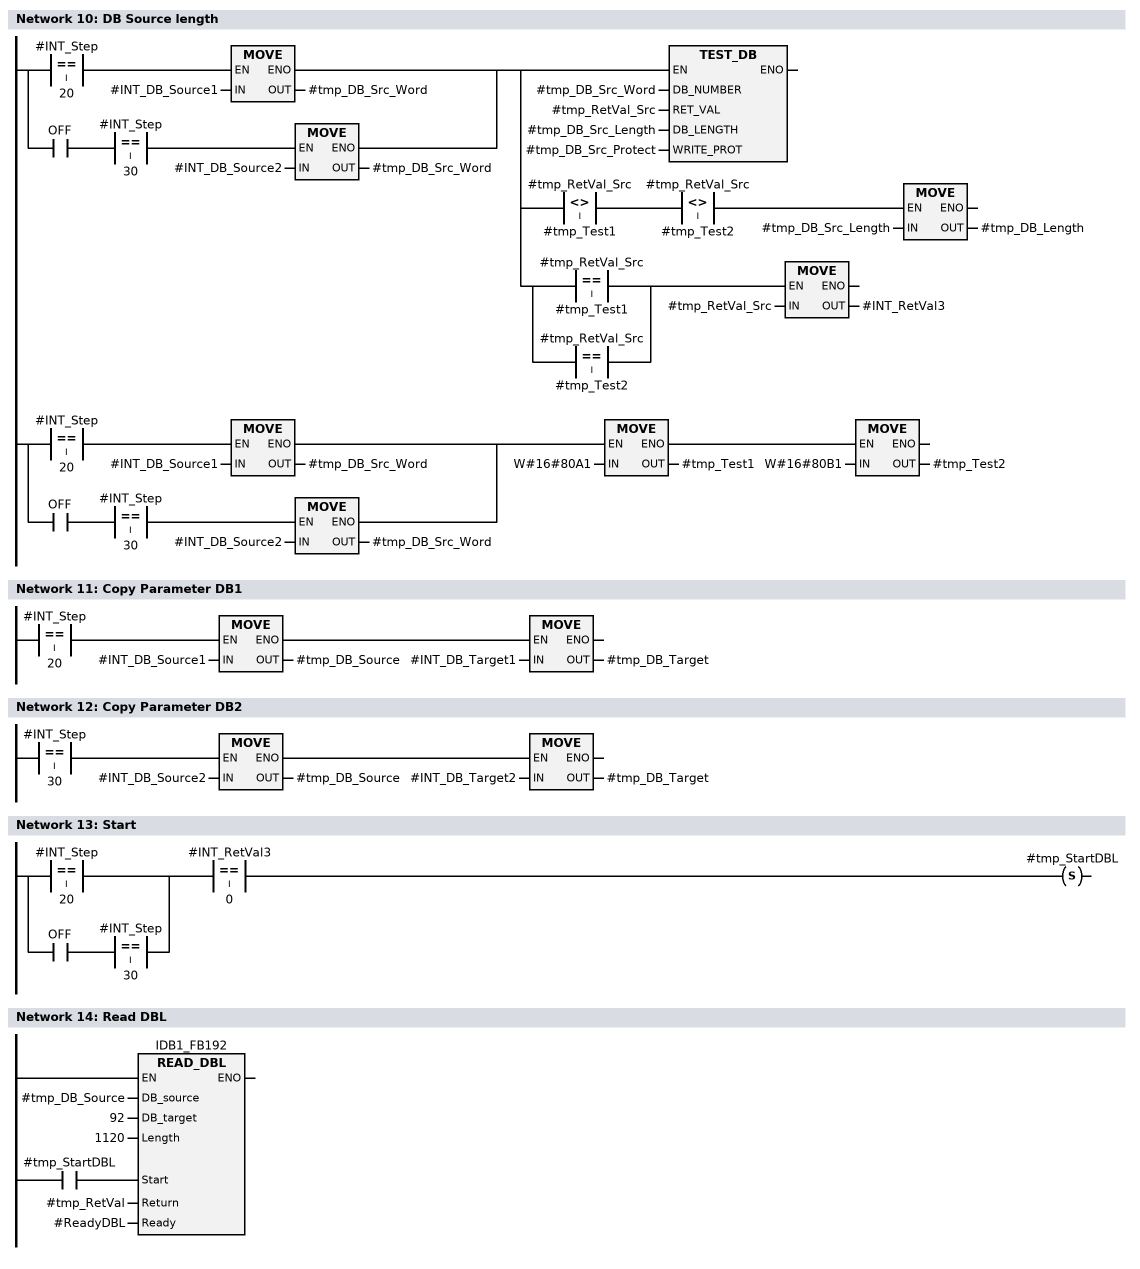
NETWORK
TITLE = DB Source length
      O(;
      A(;
      L     #INT_Step;
      L     20;
      ==I;
      );
      JNB   _00e;
      L     #INT_DB_Source1;
      T     #tmp_DB_Src_Word;
      SET;
      SAVE;
      CLR;
_00e: A     BR;
      );
      O(;
      A     "OFF";
      A(;
      L     #INT_Step;
      L     30;
      ==I;
      );
      JNB   _00f;
      L     #INT_DB_Source2;
      T     #tmp_DB_Src_Word;
      SET;
      SAVE;
      CLR;
_00f: A     BR;
      );
      =     L 16.0;
      A     L 16.0;
      JNB   _010;
      CALL  "TEST_DB" (
           DB_NUMBER                := #tmp_DB_Src_Word,
           RET_VAL                  := #tmp_RetVal_Src,
           DB_LENGTH                := #tmp_DB_Src_Length,
           WRITE_PROT               := #tmp_DB_Src_Protect);
_010: NOP   0;
      A(;
      A     L 16.0;
      JNB   _011;
      L     W#16#80A1;
      T     #tmp_Test1;
      SET;
      SAVE;
      CLR;
_011: A     BR;
      );
      JNB   _012;
      L     W#16#80B1;
      T     #tmp_Test2;
_012: NOP   0;
      A     L 16.0;
      A(;
      L     #tmp_RetVal_Src;
      L     #tmp_Test1;
      <>I;
      );
      A(;
      L     #tmp_RetVal_Src;
      L     #tmp_Test2;
      <>I;
      );
      JNB   _013;
      L     #tmp_DB_Src_Length;
      T     #tmp_DB_Length;
_013: NOP   0;
      A     L 16.0;
      A(;
      O(;
      L     #tmp_RetVal_Src;
      L     #tmp_Test1;
      ==I;
      );
      O(;
      L     #tmp_RetVal_Src;
      L     #tmp_Test2;
      ==I;
      );
      );
      JNB   _014;
      L     #tmp_RetVal_Src;
      T     #INT_RetVal3;
_014: NOP   0;
NETWORK
TITLE = Copy Parameter DB1
      A(;
      A(;
      L     #INT_Step;
      L     20;
      ==I;
      );
      JNB   _015;
      L     #INT_DB_Source1;
      T     #tmp_DB_Source;
      SET;
      SAVE;
      CLR;
_015: A     BR;
      );
      JNB   _016;
      L     #INT_DB_Target1;
      T     #tmp_DB_Target;
_016: NOP   0;
NETWORK
TITLE = Copy Parameter DB2
      A(;
      A(;
      L     #INT_Step;
      L     30;
      ==I;
      );
      JNB   _017;
      L     #INT_DB_Source2;
      T     #tmp_DB_Source;
      SET;
      SAVE;
      CLR;
_017: A     BR;
      );
      JNB   _018;
      L     #INT_DB_Target2;
      T     #tmp_DB_Target;
_018: NOP   0;
NETWORK
TITLE = Start
      A(;
      O(;
      L     #INT_Step;
      L     20;
      ==I;
      );
      O;
      A     "OFF";
      A(;
      L     #INT_Step;
      L     30;
      ==I;
      );
      );
      A(;
      L     #INT_RetVal3;
      L     0;
      ==I;
      );
      S     #tmp_StartDBL;
NETWORK
TITLE = Read DBL
      A     #tmp_StartDBL;
      =     L 16.0;
      BLD   103;
      CALL  "READ_DBL" , "IDB1_FB192" (
           DB_source                := #tmp_DB_Source,
           DB_target                := 92,
           Length                   := 1120,
           Start                    := L 16.0,
           Return                   := #tmp_RetVal,
           Ready                    := #ReadyDBL);
      NOP   0;
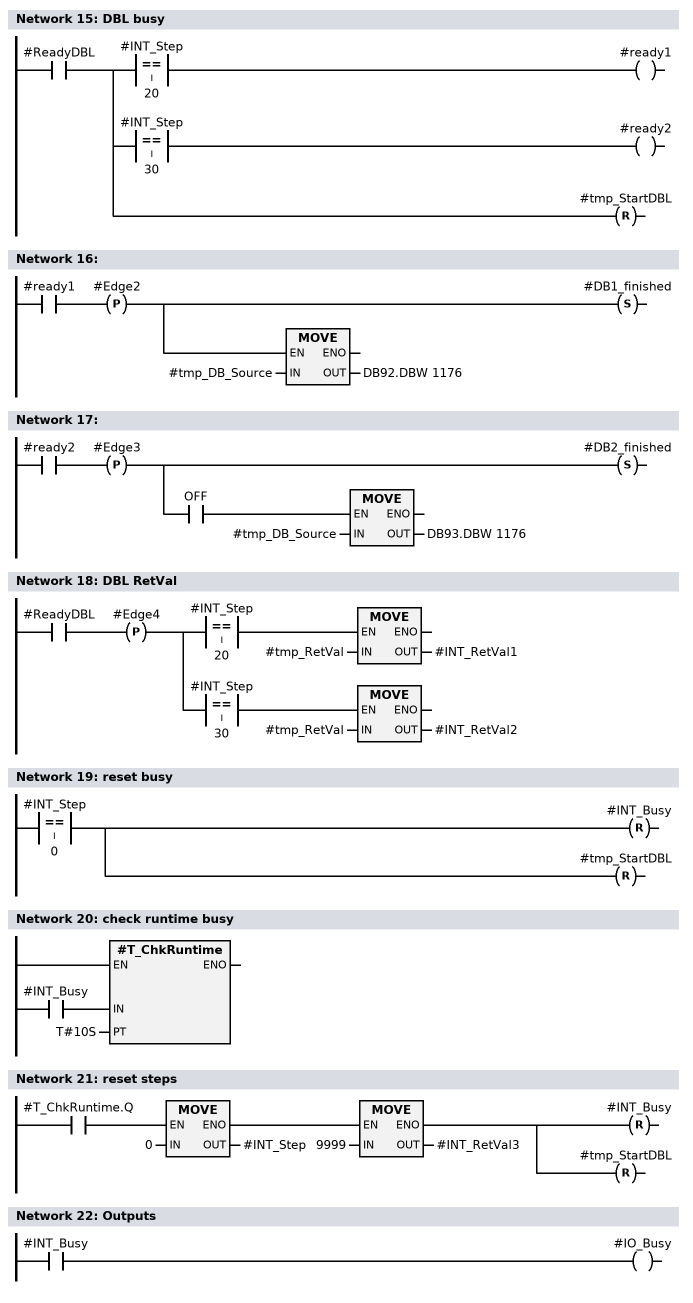
NETWORK
TITLE = DBL busy
      A     #ReadyDBL;
      =     L 16.0;
      A     L 16.0;
      A(;
      L     #INT_Step;
      L     20;
      ==I;
      );
      =     #ready1;
      A     L 16.0;
      A(;
      L     #INT_Step;
      L     30;
      ==I;
      );
      =     #ready2;
      A     L 16.0;
      BLD   102;
      R     #tmp_StartDBL;
NETWORK
TITLE =
      A     #ready1;
      BLD   100;
      FP    #Edge2;
      =     L 16.0;
      A     L 16.0;
      BLD   102;
      S     #DB1_finished;
      A     L 16.0;
      JNB   _019;
      L     #tmp_DB_Source;
      T     DB92.DBW 1176;
_019: NOP   0;
NETWORK
TITLE =
      A     #ready2;
      BLD   100;
      FP    #Edge3;
      =     L 16.0;
      A     L 16.0;
      BLD   102;
      S     #DB2_finished;
      A     L 16.0;
      A     "OFF";
      JNB   _01a;
      L     #tmp_DB_Source;
      T     DB93.DBW 1176;
_01a: NOP   0;
NETWORK
TITLE = DBL RetVal
      A     #ReadyDBL;
      BLD   100;
      FP    #Edge4;
      =     L 16.0;
      A     L 16.0;
      A(;
      L     #INT_Step;
      L     20;
      ==I;
      );
      JNB   _01b;
      L     #tmp_RetVal;
      T     #INT_RetVal1;
_01b: NOP   0;
      A     L 16.0;
      A(;
      L     #INT_Step;
      L     30;
      ==I;
      );
      JNB   _01c;
      L     #tmp_RetVal;
      T     #INT_RetVal2;
_01c: NOP   0;
NETWORK
TITLE = reset busy
      L     #INT_Step;
      L     0;
      ==I;
      R     #INT_Busy;
      R     #tmp_StartDBL;
NETWORK
TITLE = check runtime busy
      A     #INT_Busy;
      =     L 16.0;
      BLD   103;
      CALL  #T_ChkRuntime (
           IN                       := L 16.0,
           PT                       := T#10S);
      NOP   0;
NETWORK
TITLE = reset steps
      A(;
      A     #T_ChkRuntime.Q;
      JNB   _01d;
      L     0;
      T     #INT_Step;
      SET;
      SAVE;
      CLR;
_01d: A     BR;
      );
      JNB   _01e;
      L     9999;
      T     #INT_RetVal3;
      SET;
      SAVE;
      CLR;
_01e: A     BR;
      R     #INT_Busy;
      R     #tmp_StartDBL;
NETWORK
TITLE = Outputs
      A     #INT_Busy;
      =     #IO_Busy;
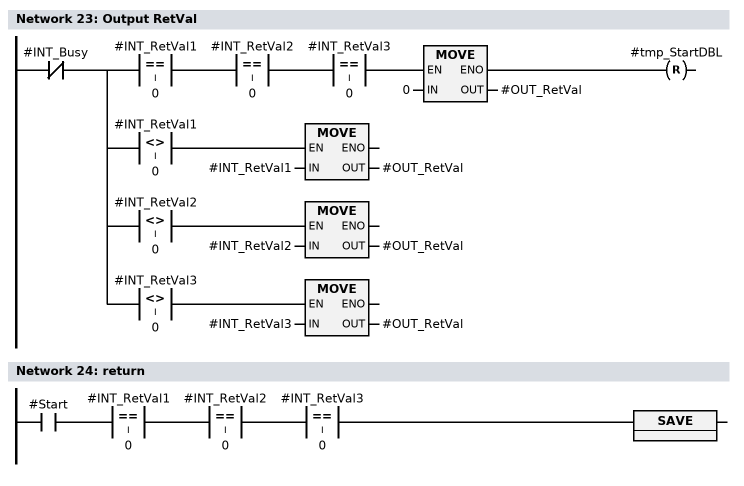
NETWORK
TITLE = Output RetVal
      AN    #INT_Busy;
      =     L 16.0;
      A     L 16.0;
      A(;
      L     #INT_RetVal1;
      L     0;
      ==I;
      );
      A(;
      L     #INT_RetVal2;
      L     0;
      ==I;
      );
      A(;
      L     #INT_RetVal3;
      L     0;
      ==I;
      );
      JNB   _01f;
      L     0;
      T     #OUT_RetVal;
      SET;
      SAVE;
      CLR;
_01f: A     BR;
      R     #tmp_StartDBL;
      A     L 16.0;
      A(;
      L     #INT_RetVal1;
      L     0;
      <>I;
      );
      JNB   _020;
      L     #INT_RetVal1;
      T     #OUT_RetVal;
_020: NOP   0;
      A     L 16.0;
      A(;
      L     #INT_RetVal2;
      L     0;
      <>I;
      );
      JNB   _021;
      L     #INT_RetVal2;
      T     #OUT_RetVal;
_021: NOP   0;
      A     L 16.0;
      A(;
      L     #INT_RetVal3;
      L     0;
      <>I;
      );
      JNB   _022;
      L     #INT_RetVal3;
      T     #OUT_RetVal;
_022: NOP   0;
NETWORK
TITLE = return
      A     #Start;
      A(;
      L     #INT_RetVal1;
      L     0;
      ==I;
      );
      A(;
      L     #INT_RetVal2;
      L     0;
      ==I;
      );
      A(;
      L     #INT_RetVal3;
      L     0;
      ==I;
      );
      SAVE;
END_FUNCTION_BLOCK

FUNCTION_BLOCK "READ_DBL"	// FB 192
TITLE = read from db on memory-card
//source-DB is on memory-card
//target-DB is on workarea of memory
VERSION : 1.0
VAR_INPUT
  DB_source : INT ;
  DB_target : INT ;
  Length : INT ;
  Start : BOOL ;
END_VAR
VAR_OUTPUT
  Return : INT ;
  Ready : BOOL ;
END_VAR
VAR
  T_Delay : SFB 4;
  INT_Cnt_Start : DINT ;
  INT_Last_State : INT ;
  INT_DB_source : INT ;
  INT_DB_target : INT ;
  INT_Length : INT ;
  Edge_Start : BOOL ;
  INT_Busy : BOOL ;
  SFC_Busy : BOOL ;
  Edge1 : BOOL ;
  Edge2 : BOOL ;
  Delay : BOOL ;
  Copy : BOOL ;
END_VAR
VAR_TEMP
  any_source : ANY ;
  any_target : ANY ;
  SysSave : UDT 2;
  INT_ON : BOOL ;
  INT_OFF : BOOL ;
  temp_return : INT ;
  startCopy : BOOL ;
END_VAR
BEGIN
NETWORK
TITLE = save register
      TAR1  #SysSave.AR1;
      TAR2  #SysSave.AR2;
      L     DBNO;
      T     #SysSave.DBNO;
      L     DINO;
      T     #SysSave.DINO;
NETWORK
TITLE = init
      SET;
      =     #INT_ON;
      CLR;
      =     #INT_OFF;
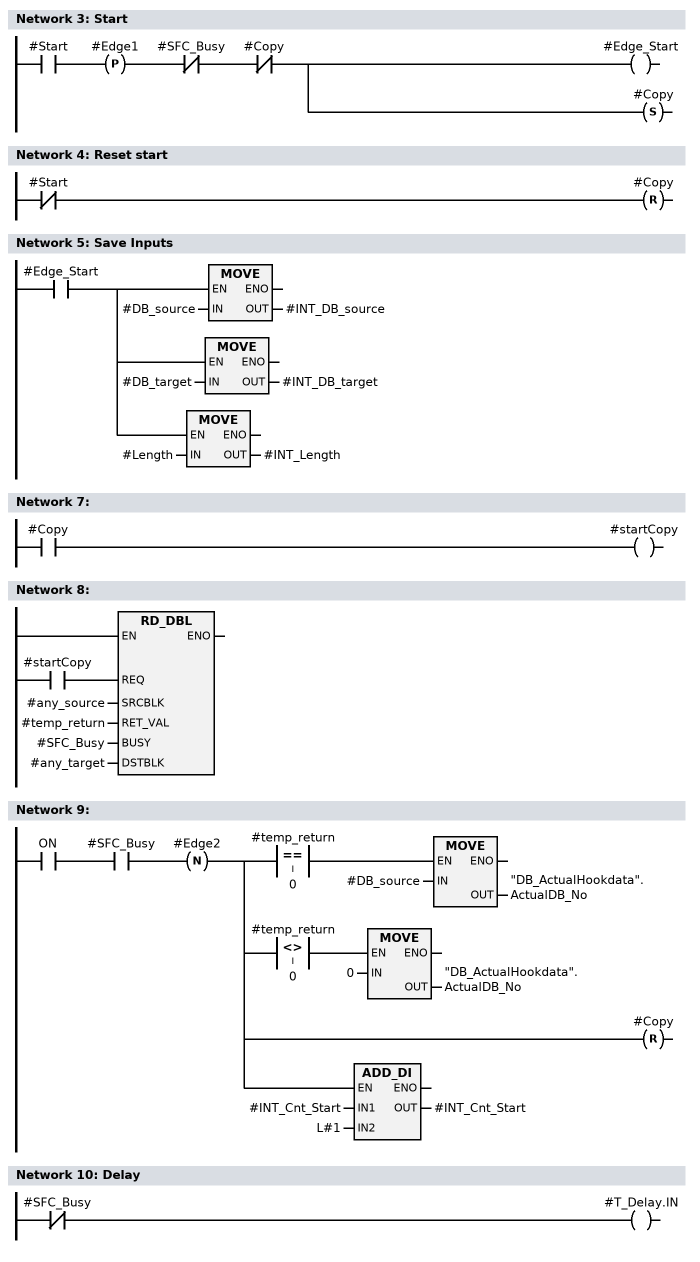
NETWORK
TITLE = Start
      A     #Start;
      FP    #Edge1;
      AN    #SFC_Busy;
      AN    #Copy;
      =     #Edge_Start;
      S     #Copy;
NETWORK
TITLE = Reset start
      AN    #Start;
      R     #Copy;
NETWORK
TITLE = Save Inputs
      A     #Edge_Start;
      =     L 37.0;
      A     L 37.0;
      JNB   _001;
      L     #DB_source;
      T     #INT_DB_source;
_001: NOP   0;
      A     L 37.0;
      JNB   _002;
      L     #DB_target;
      T     #INT_DB_target;
_002: NOP   0;
      A     L 37.0;
      JNB   _003;
      L     #Length;
      T     #INT_Length;
_003: NOP   0;
NETWORK
TITLE = create anypointer to source and target
//any to source
      L     W#16#1002;	//anytyp byte
      T     LW 0;
      L     #INT_Length;	//number of bytes
      T     LW 2;
      L     #INT_DB_source;	//number of DB-source 
      T     LW 4;
      L     0;	//begin in DB-source = byte 0
      SLD   3;
      OD    DW#16#84000000;	//constant
      T     LD 6;
//any to target
      L     W#16#1002;	//anytyp byte
      T     LW 10;
      L     #INT_Length;	//number of bytes
      T     LW 12;
      L     #INT_DB_target;	//number of DB-target
      T     LW 14;
      L     0;	//begin in DB-source = byte 0
      SLD   3;
      OD    DW#16#84000000;	//constant
      T     LD 16;
NETWORK
TITLE =
      A     #Copy;
      =     #startCopy;
NETWORK
TITLE =
      A     #startCopy;
      =     L 37.0;
      BLD   103;
      CALL  "RD_DBL" (
           REQ                      := L 37.0,
           SRCBLK                   := #any_source,
           RET_VAL                  := #temp_return,
           BUSY                     := #SFC_Busy,
           DSTBLK                   := #any_target);
      NOP   0;
NETWORK
TITLE =
//litte lazy to copy just to the end of db 92
      A     "ON";
      A(;
      A     #SFC_Busy;
      BLD   100;
      FN    #Edge2;
      );
      =     L 37.0;
      A     L 37.0;
      A(;
      L     #temp_return;
      L     0;
      ==I;
      );
      JNB   _004;
      L     #DB_source;
      T     "DB_ActualHookdata".ActualDB_No;
_004: NOP   0;
      A     L 37.0;
      A(;
      L     #temp_return;
      L     0;
      <>I;
      );
      JNB   _005;
      L     0;
      T     "DB_ActualHookdata".ActualDB_No;
_005: NOP   0;
      A     L 37.0;
      BLD   102;
      R     #Copy;
      A     L 37.0;
      JNB   _006;
      L     #INT_Cnt_Start;
      L     L#1;
      +D;
      T     #INT_Cnt_Start;
_006: NOP   0;
NETWORK
TITLE = Delay
      AN    #SFC_Busy;
      =     #T_Delay.IN;
